LIN {X 0,Y 309.605,Z 177.893,A -85,B 0,C 180,E1 -15904.089,E2 -15904.089} C_VEL
LIN {X 0,Y 309.216,Z 180.991,A -85,B 0,C 180,E1 -15904.862,E2 -15904.862} C_VEL
LIN {X 0,Y 313.855,Z 215.016,A -85,B 0,C 180,E1 -15906.096,E2 -15906.096} C_VEL
LIN {X 0,Y 315.231,Z 227.724,A -85,B 0,C 180,E1 -15906.518,E2 -15906.518} C_VEL
LIN {X 0,Y 313.627,Z 290.842,A -85,B 0,C 180,E1 -15908.084,E2 -15908.084} C_VEL
LIN {X 0,Y 312.784,Z 304.258,A -85,B 0,C 180,E1 -15908.671,E2 -15908.671} C_VEL
LIN {X 0,Y 311.715,Z 316.542,A -85,B 0,C 180,E1 -15909.459,E2 -15909.459} C_VEL
LIN {X 0,Y 310.435,Z 328.402,A -85,B 0,C 180,E1 -15910.493,E2 -15910.493} C_VEL
LIN {X 0,Y 308.971,Z 339.839,A -85,B 0,C 180,E1 -15911.774,E2 -15911.774} C_VEL
LIN {X 0,Y 307.713,Z 350.2,A -85,B 0,C 180,E1 -15913.242,E2 -15913.242} C_VEL
LIN {X 0,Y 306.659,Z 358.857,A -85,B 0,C 180,E1 -15914.757,E2 -15914.757} C_VEL
LIN {X 0,Y 305.56,Z 367.859,A -85,B 0,C 180,E1 -15916.703,E2 -15916.703} C_VEL
LIN {X 0,Y 304.589,Z 375.237,A -85,B 0,C 180,E1 -15918.689,E2 -15918.689} C_VEL
LIN {X 0,Y 304.099,Z 381.144,A -85,B 0,C 180,E1 -15920.69,E2 -15920.69} C_VEL
LIN {X 0,Y 303.823,Z 385.764,A -85,B 0,C 180,E1 -15922.691,E2 -15922.691} C_VEL
LIN {X 0,Y 303.71,Z 389.249,A -85,B 0,C 180,E1 -15924.689,E2 -15924.689} C_VEL
LIN {X 0,Y 303.749,Z 390.973,A -85,B 0,C 180,E1 -15926.02,E2 -15926.02} C_VEL
LIN {X 0,Y 303.741,Z 392.268,A -85,B 0,C 180,E1 -15927.348,E2 -15927.348} C_VEL
LIN {X 0,Y 303.826,Z 393.159,A -85,B 0,C 180,E1 -15928.674,E2 -15928.674} C_VEL
LIN {X 0,Y 303.901,Z 393.618,A -85,B 0,C 180,E1 -15930,E2 -15930} C_VEL
LIN {X 0,Y 303.777,Z 393.629,A -85,B 0,C 180,E1 -15931.326,E2 -15931.326} C_VEL
LIN {X 0,Y 303.708,Z 393.245,A -85,B 0,C 180,E1 -15932.653,E2 -15932.653} C_VEL
LIN {X 0,Y 303.702,Z 392.469,A -85,B 0,C 180,E1 -15933.981,E2 -15933.981} C_VEL
LIN {X 0,Y 303.644,Z 390.958,A -85,B 0,C 180,E1 -15935.578,E2 -15935.578} C_VEL
LIN {X 0,Y 303.882,Z 387.555,A -85,B 0,C 180,E1 -15937.976,E2 -15937.976} C_VEL
LIN {X 0,Y 304.299,Z 383.584,A -85,B 0,C 180,E1 -15939.975,E2 -15939.975} C_VEL
LIN {X 0,Y 304.977,Z 378.484,A -85,B 0,C 180,E1 -15941.97,E2 -15941.97} C_VEL
LIN {X 0,Y 306.165,Z 372.114,A -85,B 0,C 180,E1 -15943.947,E2 -15943.947} C_VEL
LIN {X 0,Y 307.574,Z 364.197,A -85,B 0,C 180,E1 -15945.914,E2 -15945.914} C_VEL
LIN {X 0,Y 309.228,Z 354.358,A -85,B 0,C 180,E1 -15947.868,E2 -15947.868} C_VEL
LIN {X 0,Y 311.011,Z 344.245,A -85,B 0,C 180,E1 -15949.47,E2 -15949.47} C_VEL
LIN {X 0,Y 312.942,Z 332.854,A -85,B 0,C 180,E1 -15950.886,E2 -15950.886} C_VEL
LIN {X 0,Y 314.607,Z 321.762,A -85,B 0,C 180,E1 -15951.973,E2 -15951.973} C_VEL
LIN {X 0,Y 316.144,Z 309.533,A -85,B 0,C 180,E1 -15952.894,E2 -15952.894} C_VEL
LIN {X 0,Y 317.465,Z 296.002,A -85,B 0,C 180,E1 -15953.608,E2 -15953.608} C_VEL
LIN {X 0,Y 318.238,Z 283.152,A -85,B 0,C 180,E1 -15954.047,E2 -15954.047} C_VEL
LIN {X 0,Y 319.862,Z 226.172,A -85,B 0,C 180,E1 -15955.466,E2 -15955.466} C_VEL
LIN {X 0,Y 317.021,Z 205.398,A -85,B 0,C 180,E1 -15956.349,E2 -15956.349} C_VEL
LIN {X 0,Y 313.131,Z 184.639,A -85,B 0,C 180,E1 -15957.383,E2 -15957.383} C_VEL
LIN {X 0,Y 311.782,Z 178.357,A -85,B 0,C 180,E1 -15957.736,E2 -15957.736} C_VEL
LIN {X 0,Y 310.59,Z 171.052,A -85,B 0,C 180,E1 -15959.855,E2 -15959.855} C_VEL
LIN {X 0,Y 308.122,Z 160.384,A -85,B 0,C 180,E1 -15963.19,E2 -15963.19} C_VEL
LIN {X 0,Y 305.482,Z 150.438,A -85,B 0,C 180,E1 -15966.587,E2 -15966.587} C_VEL
LIN {X 0,Y 305.466,Z 150.444,A -85,B 0,C 180,E1 -15970.106,E2 -15970.106} C_VEL
LIN {X 0,Y 305.447,Z 150.439,A -85,B 0,C 180,E1 -15973.651,E2 -15973.651} C_VEL
LIN {X 0,Y 305.488,Z 150.436,A -85,B 0,C 180,E1 -15977.407,E2 -15977.407} C_VEL
LIN {X 0,Y 305.518,Z 150.425,A -85,B 0,C 180,E1 -15981.603,E2 -15981.603} C_VEL
LIN {X 0,Y 305.462,Z 150.434,A -85,B 0,C 180,E1 -15984.886,E2 -15984.886} C_VEL
LIN {X 0,Y 305.452,Z 150.437,A -85,B 0,C 180,E1 -15988.354,E2 -15988.354} C_VEL
LIN {X 0,Y 305.52,Z 150.422,A -85,B 0,C 180,E1 -15991.113,E2 -15991.113} C_VEL
LIN {X 0,Y 305.57,Z 150.414,A -85,B 0,C 180,E1 -15994.087,E2 -15994.087} C_VEL
LIN {X 0,Y 305.481,Z 150.428,A -85,B 0,C 180,E1 -15998.401,E2 -15998.401} C_VEL
LIN {X 0,Y 305.589,Z 150.41,A -85,B 0,C 180,E1 -16001.217,E2 -16001.217} C_VEL
LIN {X 0,Y 305.648,Z 150.404,A -85,B 0,C 180,E1 -16005.349,E2 -16005.349} C_VEL
LIN {X 0,Y 305.637,Z 150.408,A -85,B 0,C 180,E1 -16009.399,E2 -16009.399} C_VEL
LIN {X 0,Y 305.812,Z 150.385,A -85,B 0,C 180,E1 -16012.074,E2 -16012.074} C_VEL
LIN {X 0,Y 305.688,Z 150.408,A -85,B 0,C 180,E1 -16014.723,E2 -16014.723} C_VEL
LIN {X 0,Y 305.956,Z 150.373,A -85,B 0,C 180,E1 -16018.683,E2 -16018.683} C_VEL
LIN {X 0,Y 305.956,Z 150.375,A -85,B 0,C 180,E1 -16021.316,E2 -16021.316} C_VEL
LIN {X 0,Y 305.685,Z 150.405,A -85,B 0,C 180,E1 -16025.276,E2 -16025.276} C_VEL
LIN {X 0,Y 305.795,Z 150.394,A -85,B 0,C 180,E1 -16027.926,E2 -16027.926} C_VEL
LIN {X 0,Y 305.602,Z 150.416,A -85,B 0,C 180,E1 -16031.945,E2 -16031.945} C_VEL
LIN {X 0,Y 305.636,Z 150.417,A -85,B 0,C 180,E1 -16035.035,E2 -16035.035} C_VEL
LIN {X 0,Y 305.575,Z 150.422,A -85,B 0,C 180,E1 -16039.445,E2 -16039.445} C_VEL
LIN {X 0,Y 305.527,Z 150.521,A -85,B 0,C 180,E1 -16044.062,E2 -16044.062} C_VEL
LIN {X 0,Y 306.019,Z 152.265,A -85,B 0,C 180,E1 -16044.643,E2 -16044.643} C_VEL
LIN {X 0,Y 313.705,Z 166.916,A -85,B 0,C 180,E1 -16046.023,E2 -16046.023} C_VEL
LIN {X 0,Y 320.196,Z 181.578,A -85,B 0,C 180,E1 -16047.174,E2 -16047.174} C_VEL
LIN {X 0,Y 321.198,Z 184.098,A -85,B 0,C 180,E1 -16047.354,E2 -16047.354} C_VEL
LIN {X 0,Y 318.681,Z 259.47,A -85,B 0,C 180,E1 -16049.25,E2 -16049.25} C_VEL
LIN {X 0,Y 317.9,Z 272.399,A -85,B 0,C 180,E1 -16049.829,E2 -16049.829} C_VEL
LIN {X 0,Y 316.94,Z 283.918,A -85,B 0,C 180,E1 -16050.574,E2 -16050.574} C_VEL
LIN {X 0,Y 315.772,Z 295.122,A -85,B 0,C 180,E1 -16051.535,E2 -16051.535} C_VEL
LIN {X 0,Y 314.394,Z 305.267,A -85,B 0,C 180,E1 -16052.635,E2 -16052.635} C_VEL
LIN {X 0,Y 312.641,Z 316.622,A -85,B 0,C 180,E1 -16054.193,E2 -16054.193} C_VEL
LIN {X 0,Y 310.868,Z 326.385,A -85,B 0,C 180,E1 -16055.868,E2 -16055.868} C_VEL
LIN {X 0,Y 309.235,Z 334.779,A -85,B 0,C 180,E1 -16057.68,E2 -16057.68} C_VEL
LIN {X 0,Y 307.645,Z 342.494,A -85,B 0,C 180,E1 -16059.765,E2 -16059.765} C_VEL
LIN {X 0,Y 306.527,Z 348.078,A -85,B 0,C 180,E1 -16061.675,E2 -16061.675} C_VEL
LIN {X 0,Y 305.613,Z 352.558,A -85,B 0,C 180,E1 -16063.621,E2 -16063.621} C_VEL
LIN {X 0,Y 304.652,Z 356.866,A -85,B 0,C 180,E1 -16066.206,E2 -16066.206} C_VEL
LIN {X 0,Y 304.229,Z 358.833,A -85,B 0,C 180,E1 -16067.939,E2 -16067.939} C_VEL
LIN {X 0,Y 303.894,Z 360.092,A -85,B 0,C 180,E1 -16069.744,E2 -16069.744} C_VEL
LIN {X 0,Y 303.659,Z 360.636,A -85,B 0,C 180,E1 -16071.897,E2 -16071.897} C_VEL
LIN {X 0,Y 303.648,Z 360.102,A -85,B 0,C 180,E1 -16074.104,E2 -16074.104} C_VEL
LIN {X 0,Y 303.839,Z 358.382,A -85,B 0,C 180,E1 -16076.377,E2 -16076.377} C_VEL
LIN {X 0,Y 304.229,Z 355.273,A -85,B 0,C 180,E1 -16078.73,E2 -16078.73} C_VEL
LIN {X 0,Y 304.763,Z 350.855,A -85,B 0,C 180,E1 -16081.036,E2 -16081.036} C_VEL
LIN {X 0,Y 305.446,Z 345.271,A -85,B 0,C 180,E1 -16083.215,E2 -16083.215} C_VEL
LIN {X 0,Y 306.369,Z 338.545,A -85,B 0,C 180,E1 -16085.251,E2 -16085.251} C_VEL
LIN {X 0,Y 307.411,Z 330.797,A -85,B 0,C 180,E1 -16087.13,E2 -16087.13} C_VEL
LIN {X 0,Y 308.685,Z 321.324,A -85,B 0,C 180,E1 -16088.982,E2 -16088.982} C_VEL
LIN {X 0,Y 309.814,Z 312.005,A -85,B 0,C 180,E1 -16090.452,E2 -16090.452} C_VEL
LIN {X 0,Y 311.123,Z 300.466,A -85,B 0,C 180,E1 -16091.905,E2 -16091.905} C_VEL
LIN {X 0,Y 312.261,Z 288.683,A -85,B 0,C 180,E1 -16093.071,E2 -16093.071} C_VEL
LIN {X 0,Y 313.041,Z 277.074,A -85,B 0,C 180,E1 -16093.953,E2 -16093.953} C_VEL
LIN {X 0,Y 313.833,Z 263.312,A -85,B 0,C 180,E1 -16094.692,E2 -16094.692} C_VEL
LIN {X 0,Y 314.307,Z 250.807,A -85,B 0,C 180,E1 -16095.114,E2 -16095.114} C_VEL
LIN {X 0,Y 316.167,Z 179.057,A -85,B 0,C 180,E1 -16096.847,E2 -16096.847} C_VEL
LIN {X 0,Y 308.843,Z 158.463,A -85,B 0,C 180,E1 -16097.91,E2 -16097.91} C_VEL
LIN {X 0,Y 305.699,Z 150.706,A -85,B 0,C 180,E1 -16098.353,E2 -16098.353} C_VEL
LIN {X 0,Y 305.635,Z 150.414,A -85,B 0,C 180,E1 -16098.393,E2 -16098.393} C_VEL
LIN {X 0,Y 305.8,Z 150.394,A -85,B 0,C 180,E1 -16102.074,E2 -16102.074} C_VEL
LIN {X 0,Y 305.685,Z 150.406,A -85,B 0,C 180,E1 -16104.723,E2 -16104.723} C_VEL
LIN {X 0,Y 305.955,Z 150.372,A -85,B 0,C 180,E1 -16108.684,E2 -16108.684} C_VEL
LIN {X 0,Y 305.955,Z 150.377,A -85,B 0,C 180,E1 -16111.316,E2 -16111.316} C_VEL
LIN {X 0,Y 305.674,Z 150.411,A -85,B 0,C 180,E1 -16115.277,E2 -16115.277} C_VEL
LIN {X 0,Y 305.749,Z 150.398,A -85,B 0,C 180,E1 -16117.927,E2 -16117.927} C_VEL
LIN {X 0,Y 305.599,Z 150.416,A -85,B 0,C 180,E1 -16121.945,E2 -16121.945} C_VEL
LIN {X 0,Y 305.608,Z 150.419,A -85,B 0,C 180,E1 -16125.015,E2 -16125.015} C_VEL
LIN {X 0,Y 305.541,Z 150.424,A -85,B 0,C 180,E1 -16129.426,E2 -16129.426} C_VEL
LIN {X 0,Y 305.485,Z 150.432,A -85,B 0,C 180,E1 -16133.039,E2 -16133.039} C_VEL
LIN {X 0,Y 305.553,Z 150.423,A -85,B 0,C 180,E1 -16136.229,E2 -16136.229} C_VEL
LIN {X 0,Y 305.495,Z 150.43,A -85,B 0,C 180,E1 -16139.05,E2 -16139.05} C_VEL
LIN {X 0,Y 305.464,Z 150.432,A -85,B 0,C 180,E1 -16143.517,E2 -16143.517} C_VEL
LIN {X 0,Y 305.473,Z 150.434,A -85,B 0,C 180,E1 -16146.739,E2 -16146.739} C_VEL
LIN {X 0,Y 305.453,Z 150.434,A -85,B 0,C 180,E1 -16150.6,E2 -16150.6} C_VEL
LIN {X 0,Y 305.424,Z 150.437,A -85,B 0,C 180,E1 -16153.655,E2 -16153.655} C_VEL
LIN {X 0,Y 305.453,Z 150.433,A -85,B 0,C 180,E1 -16157.414,E2 -16157.414} C_VEL
LIN {X 0,Y 305.448,Z 150.431,A -85,B 0,C 180,E1 -16161.215,E2 -16161.215} C_VEL
LIN {X 0,Y 304.815,Z 150.516,A -85,B 0,C 180,E1 -16162.315,E2 -16162.315} C_VEL
LIN {X 0,Y 301.928,Z 150.877,A -85,B 0,C 180,E1 -16164.104,E2 -16164.104} C_VEL
LIN {X 0,Y 299.474,Z 151.18,A -85,B 0,C 180,E1 -16165.556,E2 -16165.556} C_VEL
LIN {X 0,Y 298.451,Z 151.306,A -85,B 0,C 180,E1 -16166.682,E2 -16166.682} C_VEL
LIN {X 0,Y 298.386,Z 151.313,A -85,B 0,C 180,E1 -16167.063,E2 -16167.063} C_VEL
LIN {X 0,Y 298.43,Z 151.304,A -85,B 0,C 180,E1 -16170.615,E2 -16170.615} C_VEL
LIN {X 0,Y 298.482,Z 151.303,A -85,B 0,C 180,E1 -16173.474,E2 -16173.474} C_VEL
LIN {X 0,Y 298.429,Z 151.309,A -85,B 0,C 180,E1 -16176.7,E2 -16176.7} C_VEL
LIN {X 0,Y 298.537,Z 151.293,A -85,B 0,C 180,E1 -16180.757,E2 -16180.757} C_VEL
LIN {X 0,Y 298.592,Z 151.288,A -85,B 0,C 180,E1 -16184.995,E2 -16184.995} C_VEL
LIN {X 0,Y 298.593,Z 151.291,A -85,B 0,C 180,E1 -16189.147,E2 -16189.147} C_VEL
LIN {X 0,Y 298.757,Z 151.266,A -85,B 0,C 180,E1 -16191.886,E2 -16191.886} C_VEL
LIN {X 0,Y 298.659,Z 151.277,A -85,B 0,C 180,E1 -16194.599,E2 -16194.599} C_VEL
LIN {X 0,Y 298.923,Z 151.248,A -85,B 0,C 180,E1 -16198.653,E2 -16198.653} C_VEL
LIN {X 0,Y 298.923,Z 151.248,A -85,B 0,C 180,E1 -16201.348,E2 -16201.348} C_VEL
LIN {X 0,Y 298.791,Z 151.266,A -85,B 0,C 180,E1 -16206.754,E2 -16206.754} C_VEL
LIN {X 0,Y 298.68,Z 151.277,A -85,B 0,C 180,E1 -16209.481,E2 -16209.481} C_VEL
LIN {X 0,Y 298.551,Z 151.292,A -85,B 0,C 180,E1 -16213.616,E2 -16213.616} C_VEL
LIN {X 0,Y 298.548,Z 151.296,A -85,B 0,C 180,E1 -16216.409,E2 -16216.409} C_VEL
LIN {X 0,Y 298.51,Z 151.297,A -85,B 0,C 180,E1 -16219.654,E2 -16219.654} C_VEL
LIN {X 0,Y 298.428,Z 151.309,A -85,B 0,C 180,E1 -16223.6,E2 -16223.6} C_VEL
LIN {X 0,Y 298.489,Z 151.304,A -85,B 0,C 180,E1 -16226.575,E2 -16226.575} C_VEL
LIN {X 0,Y 298.421,Z 151.311,A -85,B 0,C 180,E1 -16229.641,E2 -16229.641} C_VEL
LIN {X 0,Y 298.396,Z 151.314,A -85,B 0,C 180,E1 -16232.801,E2 -16232.801} C_VEL
LIN {X 0,Y 298.466,Z 151.305,A -85,B 0,C 180,E1 -16236.813,E2 -16236.813} C_VEL
LIN {X 0,Y 298.418,Z 151.311,A -85,B 0,C 180,E1 -16241.095,E2 -16241.095} C_VEL
LIN {X 0,Y 298.427,Z 151.309,A -85,B 0,C 180,E1 -16243.109,E2 -16243.109} C_VEL
LIN {X 0,Y 298.433,Z 151.308,A -85,B 0,C 180,E1 -16246.926,E2 -16246.926} C_VEL
LIN {X 0,Y 298.432,Z 151.31,A -85,B 0,C 180,E1 -16251,E2 -16251} C_VEL
LIN {X 0,Y 298.434,Z 151.312,A -85,B 0,C 180,E1 -16253.933,E2 -16253.933} C_VEL
LIN {X 0,Y 298.472,Z 151.434,A -85,B 0,C 180,E1 -16256.099,E2 -16256.099} C_VEL
LIN {X 0,Y 301.505,Z 165.405,A -85,B 0,C 180,E1 -16260.229,E2 -16260.229} C_VEL
LIN {X 0,Y 303.03,Z 172.939,A -85,B 0,C 180,E1 -16262.364,E2 -16262.364} C_VEL
LIN {X 0,Y 302.835,Z 177.137,A -85,B 0,C 180,E1 -16263.465,E2 -16263.465} C_VEL
LIN {X 0,Y 302.407,Z 180.637,A -85,B 0,C 180,E1 -16264.362,E2 -16264.362} C_VEL
LIN {X 0,Y 307.043,Z 214.787,A -85,B 0,C 180,E1 -16265.636,E2 -16265.636} C_VEL
LIN {X 0,Y 308.549,Z 227.299,A -85,B 0,C 180,E1 -16266.074,E2 -16266.074} C_VEL
LIN {X 0,Y 306.907,Z 290.169,A -85,B 0,C 180,E1 -16267.667,E2 -16267.667} C_VEL
LIN {X 0,Y 306.041,Z 303.671,A -85,B 0,C 180,E1 -16268.266,E2 -16268.266} C_VEL
LIN {X 0,Y 304.907,Z 316.005,A -85,B 0,C 180,E1 -16269.067,E2 -16269.067} C_VEL
LIN {X 0,Y 303.528,Z 328.703,A -85,B 0,C 180,E1 -16270.206,E2 -16270.206} C_VEL
LIN {X 0,Y 302.023,Z 340.017,A -85,B 0,C 180,E1 -16271.515,E2 -16271.515} C_VEL
LIN {X 0,Y 300.732,Z 350.248,A -85,B 0,C 180,E1 -16273.015,E2 -16273.015} C_VEL
LIN {X 0,Y 299.553,Z 359.788,A -85,B 0,C 180,E1 -16274.761,E2 -16274.761} C_VEL
LIN {X 0,Y 298.406,Z 368.461,A -85,B 0,C 180,E1 -16276.725,E2 -16276.725} C_VEL
LIN {X 0,Y 297.459,Z 375.637,A -85,B 0,C 180,E1 -16278.76,E2 -16278.76} C_VEL
LIN {X 0,Y 296.946,Z 382.182,A -85,B 0,C 180,E1 -16281.151,E2 -16281.151} C_VEL
LIN {X 0,Y 296.702,Z 386.466,A -85,B 0,C 180,E1 -16283.198,E2 -16283.198} C_VEL
LIN {X 0,Y 296.642,Z 388.725,A -85,B 0,C 180,E1 -16284.562,E2 -16284.562} C_VEL
LIN {X 0,Y 296.657,Z 390.484,A -85,B 0,C 180,E1 -16285.924,E2 -16285.924} C_VEL
LIN {X 0,Y 296.661,Z 391.803,A -85,B 0,C 180,E1 -16287.284,E2 -16287.284} C_VEL
LIN {X 0,Y 296.732,Z 392.714,A -85,B 0,C 180,E1 -16288.643,E2 -16288.643} C_VEL
LIN {X 0,Y 296.811,Z 393.211,A -85,B 0,C 180,E1 -16290,E2 -16290} C_VEL
LIN {X 0,Y 296.685,Z 393.246,A -85,B 0,C 180,E1 -16291.357,E2 -16291.357} C_VEL
LIN {X 0,Y 296.628,Z 392.883,A -85,B 0,C 180,E1 -16292.716,E2 -16292.716} C_VEL
LIN {X 0,Y 296.61,Z 392.125,A -85,B 0,C 180,E1 -16294.076,E2 -16294.076} C_VEL
LIN {X 0,Y 296.547,Z 390.884,A -85,B 0,C 180,E1 -16295.508,E2 -16295.508} C_VEL
LIN {X 0,Y 296.827,Z 387.29,A -85,B 0,C 180,E1 -16298.167,E2 -16298.167} C_VEL
LIN {X 0,Y 297.269,Z 383.361,A -85,B 0,C 180,E1 -16300.213,E2 -16300.213} C_VEL
LIN {X 0,Y 297.999,Z 378.311,A -85,B 0,C 180,E1 -16302.254,E2 -16302.254} C_VEL
LIN {X 0,Y 299.262,Z 372.009,A -85,B 0,C 180,E1 -16304.275,E2 -16304.275} C_VEL
LIN {X 0,Y 300.745,Z 364.208,A -85,B 0,C 180,E1 -16306.285,E2 -16306.285} C_VEL
LIN {X 0,Y 302.141,Z 356.263,A -85,B 0,C 180,E1 -16307.951,E2 -16307.951} C_VEL
LIN {X 0,Y 304.123,Z 345.536,A -85,B 0,C 180,E1 -16309.753,E2 -16309.753} C_VEL
LIN {X 0,Y 306.153,Z 334.655,A -85,B 0,C 180,E1 -16311.195,E2 -16311.195} C_VEL
LIN {X 0,Y 308.052,Z 322.344,A -85,B 0,C 180,E1 -16312.466,E2 -16312.466} C_VEL
LIN {X 0,Y 309.805,Z 309.277,A -85,B 0,C 180,E1 -16313.479,E2 -16313.479} C_VEL
LIN {X 0,Y 311.174,Z 295.74,A -85,B 0,C 180,E1 -16314.209,E2 -16314.209} C_VEL
LIN {X 0,Y 311.981,Z 282.408,A -85,B 0,C 180,E1 -16314.674,E2 -16314.674} C_VEL
LIN {X 0,Y 313.717,Z 227.416,A -85,B 0,C 180,E1 -16316.069,E2 -16316.069} C_VEL
LIN {X 0,Y 310.987,Z 206.911,A -85,B 0,C 180,E1 -16316.971,E2 -16316.971} C_VEL
LIN {X 0,Y 307.427,Z 187.646,A -85,B 0,C 180,E1 -16317.958,E2 -16317.958} C_VEL
LIN {X 0,Y 305.766,Z 180.708,A -85,B 0,C 180,E1 -16318.374,E2 -16318.374} C_VEL
LIN {X 0,Y 304.746,Z 177.782,A -85,B 0,C 180,E1 -16318.619,E2 -16318.619} C_VEL
LIN {X 0,Y 302.538,Z 167.202,A -85,B 0,C 180,E1 -16321.903,E2 -16321.903} C_VEL
LIN {X 0,Y 300.04,Z 157.167,A -85,B 0,C 180,E1 -16325.272,E2 -16325.272} C_VEL
LIN {X 0,Y 298.434,Z 151.316,A -85,B 0,C 180,E1 -16327.423,E2 -16327.423} C_VEL
LIN {X 0,Y 298.419,Z 151.316,A -85,B 0,C 180,E1 -16331.255,E2 -16331.255} C_VEL
LIN {X 0,Y 298.36,Z 151.324,A -85,B 0,C 180,E1 -16334.964,E2 -16334.964} C_VEL
LIN {X 0,Y 298.432,Z 151.315,A -85,B 0,C 180,E1 -16336.926,E2 -16336.926} C_VEL
LIN {X 0,Y 298.431,Z 151.307,A -85,B 0,C 180,E1 -16340.999,E2 -16340.999} C_VEL
LIN {X 0,Y 298.433,Z 151.306,A -85,B 0,C 180,E1 -16343.932,E2 -16343.932} C_VEL
LIN {X 0,Y 298.395,Z 151.313,A -85,B 0,C 180,E1 -16347.983,E2 -16347.983} C_VEL
LIN {X 0,Y 298.463,Z 151.308,A -85,B 0,C 180,E1 -16351.904,E2 -16351.904} C_VEL
LIN {X 0,Y 298.483,Z 151.299,A -85,B 0,C 180,E1 -16354.923,E2 -16354.923} C_VEL
LIN {X 0,Y 298.439,Z 151.308,A -85,B 0,C 180,E1 -16359.314,E2 -16359.314} C_VEL
LIN {X 0,Y 298.537,Z 151.294,A -85,B 0,C 180,E1 -16362.179,E2 -16362.179} C_VEL
LIN {X 0,Y 298.592,Z 151.282,A -85,B 0,C 180,E1 -16364.994,E2 -16364.994} C_VEL
LIN {X 0,Y 298.592,Z 151.283,A -85,B 0,C 180,E1 -16369.146,E2 -16369.146} C_VEL
LIN {X 0,Y 298.757,Z 151.265,A -85,B 0,C 180,E1 -16371.886,E2 -16371.886} C_VEL
LIN {X 0,Y 298.659,Z 151.283,A -85,B 0,C 180,E1 -16374.599,E2 -16374.599} C_VEL
LIN {X 0,Y 298.922,Z 151.249,A -85,B 0,C 180,E1 -16378.652,E2 -16378.652} C_VEL
LIN {X 0,Y 298.922,Z 151.251,A -85,B 0,C 180,E1 -16381.347,E2 -16381.347} C_VEL
LIN {X 0,Y 298.785,Z 151.264,A -85,B 0,C 180,E1 -16386.754,E2 -16386.754} C_VEL
LIN {X 0,Y 298.634,Z 151.285,A -85,B 0,C 180,E1 -16389.482,E2 -16389.482} C_VEL
LIN {X 0,Y 298.55,Z 151.295,A -85,B 0,C 180,E1 -16393.615,E2 -16393.615} C_VEL
LIN {X 0,Y 298.547,Z 151.295,A -85,B 0,C 180,E1 -16396.408,E2 -16396.408} C_VEL
LIN {X 0,Y 298.51,Z 151.301,A -85,B 0,C 180,E1 -16399.655,E2 -16399.655} C_VEL
LIN {X 0,Y 298.494,Z 151.402,A -85,B 0,C 180,E1 -16403.26,E2 -16403.26} C_VEL
LIN {X 0,Y 298.694,Z 152.48,A -85,B 0,C 180,E1 -16403.669,E2 -16403.669} C_VEL
LIN {X 0,Y 306.611,Z 167.127,A -85,B 0,C 180,E1 -16405.181,E2 -16405.181} C_VEL
LIN {X 0,Y 312.778,Z 180.395,A -85,B 0,C 180,E1 -16406.314,E2 -16406.314} C_VEL
LIN {X 0,Y 315.128,Z 186.194,A -85,B 0,C 180,E1 -16406.75,E2 -16406.75} C_VEL
LIN {X 0,Y 312.456,Z 259.797,A -85,B 0,C 180,E1 -16408.638,E2 -16408.638} C_VEL
LIN {X 0,Y 311.609,Z 272.96,A -85,B 0,C 180,E1 -16409.24,E2 -16409.24} C_VEL
LIN {X 0,Y 310.501,Z 285.544,A -85,B 0,C 180,E1 -16410.086,E2 -16410.086} C_VEL
LIN {X 0,Y 309.168,Z 297.063,A -85,B 0,C 180,E1 -16411.129,E2 -16411.129} C_VEL
LIN {X 0,Y 307.494,Z 308.603,A -85,B 0,C 180,E1 -16412.465,E2 -16412.465} C_VEL
LIN {X 0,Y 305.806,Z 318.7,A -85,B 0,C 180,E1 -16413.939,E2 -16413.939} C_VEL
LIN {X 0,Y 304.054,Z 327.766,A -85,B 0,C 180,E1 -16415.585,E2 -16415.585} C_VEL
LIN {X 0,Y 302.35,Z 336.001,A -85,B 0,C 180,E1 -16417.435,E2 -16417.435} C_VEL
LIN {X 0,Y 300.736,Z 343.483,A -85,B 0,C 180,E1 -16419.54,E2 -16419.54} C_VEL
LIN {X 0,Y 299.378,Z 349.659,A -85,B 0,C 180,E1 -16421.795,E2 -16421.795} C_VEL
LIN {X 0,Y 298.329,Z 354.37,A -85,B 0,C 180,E1 -16424.068,E2 -16424.068} C_VEL
LIN {X 0,Y 297.418,Z 358.234,A -85,B 0,C 180,E1 -16426.744,E2 -16426.744} C_VEL
LIN {X 0,Y 296.875,Z 360.309,A -85,B 0,C 180,E1 -16429.248,E2 -16429.248} C_VEL
LIN {X 0,Y 296.581,Z 361.042,A -85,B 0,C 180,E1 -16431.967,E2 -16431.967} C_VEL
LIN {X 0,Y 296.553,Z 360.638,A -85,B 0,C 180,E1 -16433.684,E2 -16433.684} C_VEL
LIN {X 0,Y 296.692,Z 359.105,A -85,B 0,C 180,E1 -16436.003,E2 -16436.003} C_VEL
LIN {X 0,Y 297.114,Z 355.879,A -85,B 0,C 180,E1 -16438.642,E2 -16438.642} C_VEL
LIN {X 0,Y 297.647,Z 351.78,A -85,B 0,C 180,E1 -16440.884,E2 -16440.884} C_VEL
LIN {X 0,Y 298.423,Z 345.503,A -85,B 0,C 180,E1 -16443.419,E2 -16443.419} C_VEL
LIN {X 0,Y 299.46,Z 338.296,A -85,B 0,C 180,E1 -16445.617,E2 -16445.617} C_VEL
LIN {X 0,Y 300.658,Z 329.79,A -85,B 0,C 180,E1 -16447.676,E2 -16447.676} C_VEL
LIN {X 0,Y 301.797,Z 321.404,A -85,B 0,C 180,E1 -16449.316,E2 -16449.316} C_VEL
LIN {X 0,Y 303.032,Z 311.571,A -85,B 0,C 180,E1 -16450.878,E2 -16450.878} C_VEL
LIN {X 0,Y 304.394,Z 299.598,A -85,B 0,C 180,E1 -16452.392,E2 -16452.392} C_VEL
LIN {X 0,Y 305.566,Z 287.769,A -85,B 0,C 180,E1 -16453.55,E2 -16453.55} C_VEL
LIN {X 0,Y 306.407,Z 275.87,A -85,B 0,C 180,E1 -16454.438,E2 -16454.438} C_VEL
LIN {X 0,Y 307.155,Z 262.7,A -85,B 0,C 180,E1 -16455.138,E2 -16455.138} C_VEL
LIN {X 0,Y 307.641,Z 249.064,A -85,B 0,C 180,E1 -16455.577,E2 -16455.577} C_VEL
LIN {X 0,Y 309.367,Z 180.053,A -85,B 0,C 180,E1 -16457.291,E2 -16457.291} C_VEL
LIN {X 0,Y 302.107,Z 159.981,A -85,B 0,C 180,E1 -16458.369,E2 -16458.369} C_VEL
LIN {X 0,Y 298.761,Z 152.111,A -85,B 0,C 180,E1 -16458.844,E2 -16458.844} C_VEL
LIN {X 0,Y 298.612,Z 151.29,A -85,B 0,C 180,E1 -16458.916,E2 -16458.916} C_VEL
LIN {X 0,Y 298.745,Z 151.274,A -85,B 0,C 180,E1 -16461.886,E2 -16461.886} C_VEL
LIN {X 0,Y 298.656,Z 151.282,A -85,B 0,C 180,E1 -16464.599,E2 -16464.599} C_VEL
LIN {X 0,Y 298.922,Z 151.248,A -85,B 0,C 180,E1 -16468.653,E2 -16468.653} C_VEL
LIN {X 0,Y 298.922,Z 151.253,A -85,B 0,C 180,E1 -16471.347,E2 -16471.347} C_VEL
LIN {X 0,Y 298.642,Z 151.287,A -85,B 0,C 180,E1 -16475.401,E2 -16475.401} C_VEL
LIN {X 0,Y 298.708,Z 151.277,A -85,B 0,C 180,E1 -16478.821,E2 -16478.821} C_VEL
LIN {X 0,Y 298.545,Z 151.295,A -85,B 0,C 180,E1 -16483.616,E2 -16483.616} C_VEL
LIN {X 0,Y 298.486,Z 151.303,A -85,B 0,C 180,E1 -16486.412,E2 -16486.412} C_VEL
LIN {X 0,Y 298.482,Z 151.302,A -85,B 0,C 180,E1 -16489.639,E2 -16489.639} C_VEL
LIN {X 0,Y 298.428,Z 151.308,A -85,B 0,C 180,E1 -16493.6,E2 -16493.6} C_VEL
LIN {X 0,Y 298.491,Z 151.305,A -85,B 0,C 180,E1 -16496.574,E2 -16496.574} C_VEL
LIN {X 0,Y 298.42,Z 151.31,A -85,B 0,C 180,E1 -16499.641,E2 -16499.641} C_VEL
LIN {X 0,Y 298.394,Z 151.316,A -85,B 0,C 180,E1 -16502.8,E2 -16502.8} C_VEL
LIN {X 0,Y 298.445,Z 151.309,A -85,B 0,C 180,E1 -16506.808,E2 -16506.808} C_VEL
LIN {X 0,Y 298.385,Z 151.311,A -85,B 0,C 180,E1 -16511.088,E2 -16511.088} C_VEL
LIN {X 0,Y 298.397,Z 151.312,A -85,B 0,C 180,E1 -16513.103,E2 -16513.103} C_VEL
LIN {X 0,Y 298.401,Z 151.312,A -85,B 0,C 180,E1 -16516.921,E2 -16516.921} C_VEL
LIN {X 0,Y 298.406,Z 151.308,A -85,B 0,C 180,E1 -16521.207,E2 -16521.207} C_VEL
LIN {X 0,Y 298.419,Z 151.313,A -85,B 0,C 180,E1 -16523.931,E2 -16523.931} C_VEL
LIN {X 0,Y 298.386,Z 151.313,A -85,B 0,C 180,E1 -16527.063,E2 -16527.063} C_VEL
LIN {X 0,Y 297.763,Z 151.396,A -85,B 0,C 180,E1 -16528.19,E2 -16528.19} C_VEL
LIN {X 0,Y 294.92,Z 151.748,A -85,B 0,C 180,E1 -16530.026,E2 -16530.026} C_VEL
LIN {X 0,Y 292.503,Z 152.045,A -85,B 0,C 180,E1 -16531.516,E2 -16531.516} C_VEL
LIN {X 0,Y 291.497,Z 152.17,A -85,B 0,C 180,E1 -16532.67,E2 -16532.67} C_VEL
LIN {X 0,Y 291.434,Z 152.178,A -85,B 0,C 180,E1 -16533.061,E2 -16533.061} C_VEL
LIN {X 0,Y 291.373,Z 152.19,A -85,B 0,C 180,E1 -16537.299,E2 -16537.299} C_VEL
LIN {X 0,Y 291.457,Z 152.175,A -85,B 0,C 180,E1 -16540.27,E2 -16540.27} C_VEL
LIN {X 0,Y 291.554,Z 152.163,A -85,B 0,C 180,E1 -16544.624,E2 -16544.624} C_VEL
LIN {X 0,Y 291.536,Z 152.168,A -85,B 0,C 180,E1 -16548.881,E2 -16548.881} C_VEL
LIN {X 0,Y 291.708,Z 152.144,A -85,B 0,C 180,E1 -16551.689,E2 -16551.689} C_VEL
LIN {X 0,Y 291.63,Z 152.152,A -85,B 0,C 180,E1 -16554.469,E2 -16554.469} C_VEL
LIN {X 0,Y 291.889,Z 152.124,A -85,B 0,C 180,E1 -16558.621,E2 -16558.621} C_VEL
LIN {X 0,Y 291.889,Z 152.123,A -85,B 0,C 180,E1 -16561.38,E2 -16561.38} C_VEL
LIN {X 0,Y 291.74,Z 152.145,A -85,B 0,C 180,E1 -16566.918,E2 -16566.918} C_VEL
LIN {X 0,Y 291.629,Z 152.155,A -85,B 0,C 180,E1 -16569.712,E2 -16569.712} C_VEL
LIN {X 0,Y 291.521,Z 152.168,A -85,B 0,C 180,E1 -16573.951,E2 -16573.951} C_VEL
LIN {X 0,Y 291.487,Z 152.177,A -85,B 0,C 180,E1 -16576.818,E2 -16576.818} C_VEL
LIN {X 0,Y 291.45,Z 152.176,A -85,B 0,C 180,E1 -16579.875,E2 -16579.875} C_VEL
LIN {X 0,Y 291.383,Z 152.189,A -85,B 0,C 180,E1 -16584.207,E2 -16584.207} C_VEL
LIN {X 0,Y 291.423,Z 152.181,A -85,B 0,C 180,E1 -16587.272,E2 -16587.272} C_VEL
LIN {X 0,Y 291.337,Z 152.196,A -85,B 0,C 180,E1 -16590.437,E2 -16590.437} C_VEL
LIN {X 0,Y 291.345,Z 152.192,A -85,B 0,C 180,E1 -16593.699,E2 -16593.699} C_VEL
LIN {X 0,Y 291.401,Z 152.184,A -85,B 0,C 180,E1 -16597.261,E2 -16597.261} C_VEL
LIN {X 0,Y 291.377,Z 152.189,A -85,B 0,C 180,E1 -16600.635,E2 -16600.635} C_VEL
LIN {X 0,Y 291.302,Z 152.198,A -85,B 0,C 180,E1 -16604.4,E2 -16604.4} C_VEL
LIN {X 0,Y 291.356,Z 152.192,A -85,B 0,C 180,E1 -16608.398,E2 -16608.398} C_VEL
LIN {X 0,Y 291.382,Z 152.189,A -85,B 0,C 180,E1 -16611.163,E2 -16611.163} C_VEL
LIN {X 0,Y 291.387,Z 152.188,A -85,B 0,C 180,E1 -16614.63,E2 -16614.63} C_VEL
LIN {X 0,Y 291.409,Z 152.396,A -85,B 0,C 180,E1 -16615.705,E2 -16615.705} C_VEL
LIN {X 0,Y 294.05,Z 164.401,A -85,B 0,C 180,E1 -16619.365,E2 -16619.365} C_VEL
LIN {X 0,Y 295.946,Z 173.524,A -85,B 0,C 180,E1 -16622.03,E2 -16622.03} C_VEL
LIN {X 0,Y 296.103,Z 176.358,A -85,B 0,C 180,E1 -16622.813,E2 -16622.813} C_VEL
LIN {X 0,Y 295.599,Z 180.238,A -85,B 0,C 180,E1 -16623.83,E2 -16623.83} C_VEL
LIN {X 0,Y 300.386,Z 215.514,A -85,B 0,C 180,E1 -16625.192,E2 -16625.192} C_VEL
LIN {X 0,Y 301.821,Z 228.349,A -85,B 0,C 180,E1 -16625.646,E2 -16625.646} C_VEL
LIN {X 0,Y 300.191,Z 289.491,A -85,B 0,C 180,E1 -16627.231,E2 -16627.231} C_VEL
LIN {X 0,Y 299.302,Z 303.08,A -85,B 0,C 180,E1 -16627.842,E2 -16627.842} C_VEL
LIN {X 0,Y 298.145,Z 315.473,A -85,B 0,C 180,E1 -16628.66,E2 -16628.66} C_VEL
LIN {X 0,Y 296.806,Z 327.414,A -85,B 0,C 180,E1 -16629.739,E2 -16629.739} C_VEL
LIN {X 0,Y 295.306,Z 338.902,A -85,B 0,C 180,E1 -16631.079,E2 -16631.079} C_VEL
LIN {X 0,Y 293.918,Z 349.293,A -85,B 0,C 180,E1 -16632.609,E2 -16632.609} C_VEL
LIN {X 0,Y 292.593,Z 359.147,A -85,B 0,C 180,E1 -16634.436,E2 -16634.436} C_VEL
LIN {X 0,Y 291.462,Z 367.691,A -85,B 0,C 180,E1 -16636.402,E2 -16636.402} C_VEL
LIN {X 0,Y 290.451,Z 374.958,A -85,B 0,C 180,E1 -16638.485,E2 -16638.485} C_VEL
LIN {X 0,Y 290.018,Z 379.867,A -85,B 0,C 180,E1 -16640.234,E2 -16640.234} C_VEL
LIN {X 0,Y 289.698,Z 384.607,A -85,B 0,C 180,E1 -16642.332,E2 -16642.332} C_VEL
LIN {X 0,Y 289.56,Z 388.19,A -85,B 0,C 180,E1 -16644.429,E2 -16644.429} C_VEL
LIN {X 0,Y 289.57,Z 389.995,A -85,B 0,C 180,E1 -16645.824,E2 -16645.824} C_VEL
LIN {X 0,Y 289.583,Z 391.337,A -85,B 0,C 180,E1 -16647.218,E2 -16647.218} C_VEL
LIN {X 0,Y 289.64,Z 392.269,A -85,B 0,C 180,E1 -16648.61,E2 -16648.61} C_VEL
LIN {X 0,Y 289.721,Z 392.796,A -85,B 0,C 180,E1 -16650,E2 -16650} C_VEL
LIN {X 0,Y 289.595,Z 392.864,A -85,B 0,C 180,E1 -16651.391,E2 -16651.391} C_VEL
LIN {X 0,Y 289.55,Z 392.521,A -85,B 0,C 180,E1 -16652.782,E2 -16652.782} C_VEL
LIN {X 0,Y 289.521,Z 391.781,A -85,B 0,C 180,E1 -16654.176,E2 -16654.176} C_VEL
LIN {X 0,Y 289.477,Z 390.642,A -85,B 0,C 180,E1 -16655.573,E2 -16655.573} C_VEL
LIN {X 0,Y 289.653,Z 388.11,A -85,B 0,C 180,E1 -16657.669,E2 -16657.669} C_VEL
LIN {X 0,Y 290.056,Z 384.584,A -85,B 0,C 180,E1 -16659.765,E2 -16659.765} C_VEL
LIN {X 0,Y 290.717,Z 379.981,A -85,B 0,C 180,E1 -16661.858,E2 -16661.858} C_VEL
LIN {X 0,Y 292.123,Z 373.074,A -85,B 0,C 180,E1 -16664.276,E2 -16664.276} C_VEL
LIN {X 0,Y 293.625,Z 365.59,A -85,B 0,C 180,E1 -16666.334,E2 -16666.334} C_VEL
LIN {X 0,Y 295.372,Z 356.355,A -85,B 0,C 180,E1 -16668.377,E2 -16668.377} C_VEL
LIN {X 0,Y 297.471,Z 345.736,A -85,B 0,C 180,E1 -16670.214,E2 -16670.214} C_VEL
LIN {X 0,Y 299.573,Z 334.994,A -85,B 0,C 180,E1 -16671.684,E2 -16671.684} C_VEL
LIN {X 0,Y 301.261,Z 324.692,A -85,B 0,C 180,E1 -16672.82,E2 -16672.82} C_VEL
LIN {X 0,Y 303.083,Z 312.471,A -85,B 0,C 180,E1 -16673.85,E2 -16673.85} C_VEL
LIN {X 0,Y 304.652,Z 299.098,A -85,B 0,C 180,E1 -16674.67,E2 -16674.67} C_VEL
LIN {X 0,Y 305.602,Z 286.943,A -85,B 0,C 180,E1 -16675.179,E2 -16675.179} C_VEL
LIN {X 0,Y 307.61,Z 228.504,A -85,B 0,C 180,E1 -16676.709,E2 -16676.709} C_VEL
LIN {X 0,Y 305.105,Z 209.128,A -85,B 0,C 180,E1 -16677.583,E2 -16677.583} C_VEL
LIN {X 0,Y 301.532,Z 189.288,A -85,B 0,C 180,E1 -16678.636,E2 -16678.636} C_VEL
LIN {X 0,Y 300.03,Z 183.283,A -85,B 0,C 180,E1 -16679.019,E2 -16679.019} C_VEL
LIN {X 0,Y 297.514,Z 177.177,A -85,B 0,C 180,E1 -16679.597,E2 -16679.597} C_VEL
LIN {X 0,Y 295.432,Z 167.395,A -85,B 0,C 180,E1 -16682.765,E2 -16682.765} C_VEL
LIN {X 0,Y 292.76,Z 157.054,A -85,B 0,C 180,E1 -16686.41,E2 -16686.41} C_VEL
LIN {X 0,Y 291.392,Z 152.195,A -85,B 0,C 180,E1 -16688.31,E2 -16688.31} C_VEL
LIN {X 0,Y 291.351,Z 152.199,A -85,B 0,C 180,E1 -16692.486,E2 -16692.486} C_VEL
LIN {X 0,Y 291.33,Z 152.197,A -85,B 0,C 180,E1 -16696.362,E2 -16696.362} C_VEL
LIN {X 0,Y 291.398,Z 152.185,A -85,B 0,C 180,E1 -16700.514,E2 -16700.514} C_VEL
LIN {X 0,Y 291.433,Z 152.183,A -85,B 0,C 180,E1 -16702.923,E2 -16702.923} C_VEL
LIN {X 0,Y 291.345,Z 152.191,A -85,B 0,C 180,E1 -16706.301,E2 -16706.301} C_VEL
LIN {X 0,Y 291.386,Z 152.181,A -85,B 0,C 180,E1 -16710.26,E2 -16710.26} C_VEL
LIN {X 0,Y 291.415,Z 152.177,A -85,B 0,C 180,E1 -16714.271,E2 -16714.271} C_VEL
LIN {X 0,Y 291.373,Z 152.18,A -85,B 0,C 180,E1 -16717.299,E2 -16717.299} C_VEL
LIN {X 0,Y 291.457,Z 152.173,A -85,B 0,C 180,E1 -16720.27,E2 -16720.27} C_VEL
LIN {X 0,Y 291.554,Z 152.158,A -85,B 0,C 180,E1 -16724.623,E2 -16724.623} C_VEL
LIN {X 0,Y 291.536,Z 152.161,A -85,B 0,C 180,E1 -16728.88,E2 -16728.88} C_VEL
LIN {X 0,Y 291.708,Z 152.144,A -85,B 0,C 180,E1 -16731.688,E2 -16731.688} C_VEL
LIN {X 0,Y 291.629,Z 152.158,A -85,B 0,C 180,E1 -16734.468,E2 -16734.468} C_VEL
LIN {X 0,Y 291.888,Z 152.126,A -85,B 0,C 180,E1 -16738.62,E2 -16738.62} C_VEL
LIN {X 0,Y 291.888,Z 152.127,A -85,B 0,C 180,E1 -16741.379,E2 -16741.379} C_VEL
LIN {X 0,Y 291.733,Z 152.143,A -85,B 0,C 180,E1 -16746.918,E2 -16746.918} C_VEL
LIN {X 0,Y 291.573,Z 152.166,A -85,B 0,C 180,E1 -16749.713,E2 -16749.713} C_VEL
LIN {X 0,Y 291.52,Z 152.17,A -85,B 0,C 180,E1 -16753.95,E2 -16753.95} C_VEL
LIN {X 0,Y 291.485,Z 152.177,A -85,B 0,C 180,E1 -16756.818,E2 -16756.818} C_VEL
LIN {X 0,Y 291.455,Z 152.18,A -85,B 0,C 180,E1 -16759.878,E2 -16759.878} C_VEL
LIN {X 0,Y 291.427,Z 152.399,A -85,B 0,C 180,E1 -16762.416,E2 -16762.416} C_VEL
LIN {X 0,Y 291.583,Z 153.109,A -85,B 0,C 180,E1 -16762.684,E2 -16762.684} C_VEL
LIN {X 0,Y 293,Z 155.84,A -85,B 0,C 180,E1 -16762.986,E2 -16762.986} C_VEL
LIN {X 0,Y 299.75,Z 167.662,A -85,B 0,C 180,E1 -16764.312,E2 -16764.312} C_VEL
LIN {X 0,Y 305.44,Z 179.616,A -85,B 0,C 180,E1 -16765.421,E2 -16765.421} C_VEL
LIN {X 0,Y 308.979,Z 187.96,A -85,B 0,C 180,E1 -16766.099,E2 -16766.099} C_VEL
LIN {X 0,Y 306.285,Z 260.08,A -85,B 0,C 180,E1 -16767.99,E2 -16767.99} C_VEL
LIN {X 0,Y 305.358,Z 273.453,A -85,B 0,C 180,E1 -16768.609,E2 -16768.609} C_VEL
LIN {X 0,Y 304.185,Z 286.327,A -85,B 0,C 180,E1 -16769.499,E2 -16769.499} C_VEL
LIN {X 0,Y 302.752,Z 298.029,A -85,B 0,C 180,E1 -16770.591,E2 -16770.591} C_VEL
LIN {X 0,Y 301.182,Z 308.317,A -85,B 0,C 180,E1 -16771.806,E2 -16771.806} C_VEL
LIN {X 0,Y 299.444,Z 318.279,A -85,B 0,C 180,E1 -16773.268,E2 -16773.268} C_VEL
LIN {X 0,Y 297.661,Z 327.265,A -85,B 0,C 180,E1 -16774.896,E2 -16774.896} C_VEL
LIN {X 0,Y 295.823,Z 335.637,A -85,B 0,C 180,E1 -16776.775,E2 -16776.775} C_VEL
LIN {X 0,Y 294.214,Z 342.701,A -85,B 0,C 180,E1 -16778.749,E2 -16778.749} C_VEL
LIN {X 0,Y 292.709,Z 349.249,A -85,B 0,C 180,E1 -16781.075,E2 -16781.075} C_VEL
LIN {X 0,Y 291.436,Z 354.616,A -85,B 0,C 180,E1 -16783.66,E2 -16783.66} C_VEL
LIN {X 0,Y 290.749,Z 357.432,A -85,B 0,C 180,E1 -16785.494,E2 -16785.494} C_VEL
LIN {X 0,Y 290.188,Z 359.453,A -85,B 0,C 180,E1 -16787.303,E2 -16787.303} C_VEL
LIN {X 0,Y 289.839,Z 360.732,A -85,B 0,C 180,E1 -16789.104,E2 -16789.104} C_VEL
LIN {X 0,Y 289.597,Z 361.375,A -85,B 0,C 180,E1 -16790.948,E2 -16790.948} C_VEL
LIN {X 0,Y 289.449,Z 361.171,A -85,B 0,C 180,E1 -16793.25,E2 -16793.25} C_VEL
LIN {X 0,Y 289.588,Z 359.821,A -85,B 0,C 180,E1 -16795.603,E2 -16795.603} C_VEL
LIN {X 0,Y 289.909,Z 357.174,A -85,B 0,C 180,E1 -16798.046,E2 -16798.046} C_VEL
LIN {X 0,Y 290.481,Z 353.016,A -85,B 0,C 180,E1 -16800.574,E2 -16800.574} C_VEL
LIN {X 0,Y 291.072,Z 348.25,A -85,B 0,C 180,E1 -16802.693,E2 -16802.693} C_VEL
LIN {X 0,Y 292.092,Z 341.199,A -85,B 0,C 180,E1 -16805.098,E2 -16805.098} C_VEL
LIN {X 0,Y 293.138,Z 333.902,A -85,B 0,C 180,E1 -16807.071,E2 -16807.071} C_VEL
LIN {X 0,Y 294.447,Z 324.905,A -85,B 0,C 180,E1 -16809.021,E2 -16809.021} C_VEL
LIN {X 0,Y 295.825,Z 314.486,A -85,B 0,C 180,E1 -16810.826,E2 -16810.826} C_VEL
LIN {X 0,Y 297.123,Z 304.077,A -85,B 0,C 180,E1 -16812.27,E2 -16812.27} C_VEL
LIN {X 0,Y 298.403,Z 291.994,A -85,B 0,C 180,E1 -16813.583,E2 -16813.583} C_VEL
LIN {X 0,Y 299.402,Z 279.714,A -85,B 0,C 180,E1 -16814.61,E2 -16814.61} C_VEL
LIN {X 0,Y 300.229,Z 266.893,A -85,B 0,C 180,E1 -16815.382,E2 -16815.382} C_VEL
LIN {X 0,Y 300.773,Z 254.043,A -85,B 0,C 180,E1 -16815.884,E2 -16815.884} C_VEL
LIN {X 0,Y 302.842,Z 181.914,A -85,B 0,C 180,E1 -16817.712,E2 -16817.712} C_VEL
LIN {X 0,Y 295.811,Z 162.524,A -85,B 0,C 180,E1 -16818.783,E2 -16818.783} C_VEL
LIN {X 0,Y 291.678,Z 152.824,A -85,B 0,C 180,E1 -16819.392,E2 -16819.392} C_VEL
LIN {X 0,Y 291.557,Z 152.172,A -85,B 0,C 180,E1 -16819.427,E2 -16819.427} C_VEL
LIN {X 0,Y 291.737,Z 152.147,A -85,B 0,C 180,E1 -16823.082,E2 -16823.082} C_VEL
LIN {X 0,Y 291.888,Z 152.124,A -85,B 0,C 180,E1 -16828.62,E2 -16828.62} C_VEL
LIN {X 0,Y 291.888,Z 152.129,A -85,B 0,C 180,E1 -16831.38,E2 -16831.38} C_VEL
LIN {X 0,Y 291.61,Z 152.162,A -85,B 0,C 180,E1 -16835.532,E2 -16835.532} C_VEL
LIN {X 0,Y 291.667,Z 152.155,A -85,B 0,C 180,E1 -16838.911,E2 -16838.911} C_VEL
LIN {X 0,Y 291.516,Z 152.172,A -85,B 0,C 180,E1 -16842.531,E2 -16842.531} C_VEL
LIN {X 0,Y 291.506,Z 152.173,A -85,B 0,C 180,E1 -16845.379,E2 -16845.379} C_VEL
LIN {X 0,Y 291.423,Z 152.181,A -85,B 0,C 180,E1 -16849.86,E2 -16849.86} C_VEL
LIN {X 0,Y 291.382,Z 152.187,A -85,B 0,C 180,E1 -16854.207,E2 -16854.207} C_VEL
LIN {X 0,Y 291.425,Z 152.181,A -85,B 0,C 180,E1 -16857.271,E2 -16857.271} C_VEL
LIN {X 0,Y 291.337,Z 152.196,A -85,B 0,C 180,E1 -16860.437,E2 -16860.437} C_VEL
LIN {X 0,Y 291.344,Z 152.192,A -85,B 0,C 180,E1 -16863.698,E2 -16863.698} C_VEL
LIN {X 0,Y 291.375,Z 152.188,A -85,B 0,C 180,E1 -16867.254,E2 -16867.254} C_VEL
LIN {X 0,Y 291.331,Z 152.192,A -85,B 0,C 180,E1 -16870.643,E2 -16870.643} C_VEL
LIN {X 0,Y 291.289,Z 152.202,A -85,B 0,C 180,E1 -16874.402,E2 -16874.402} C_VEL
LIN {X 0,Y 291.325,Z 152.194,A -85,B 0,C 180,E1 -16878.404,E2 -16878.404} C_VEL
LIN {X 0,Y 291.362,Z 152.185,A -85,B 0,C 180,E1 -16881.16,E2 -16881.16} C_VEL
LIN {X 0,Y 291.361,Z 152.19,A -85,B 0,C 180,E1 -16884.626,E2 -16884.626} C_VEL
LIN {X 0,Y 291.371,Z 152.19,A -85,B 0,C 180,E1 -16887.951,E2 -16887.951} C_VEL
LIN {X 0,Y 291.38,Z 152.182,A -85,B 0,C 180,E1 -16891.158,E2 -16891.158} C_VEL
LIN {X 0,Y 291.434,Z 152.178,A -85,B 0,C 180,E1 -16893.061,E2 -16893.061} C_VEL
LIN {X 0,Y 290.795,Z 152.263,A -85,B 0,C 180,E1 -16894.214,E2 -16894.214} C_VEL
LIN {X 0,Y 287.89,Z 152.624,A -85,B 0,C 180,E1 -16896.09,E2 -16896.09} C_VEL
LIN {X 0,Y 285.421,Z 152.934,A -85,B 0,C 180,E1 -16897.613,E2 -16897.613} C_VEL
LIN {X 0,Y 284.395,Z 153.056,A -85,B 0,C 180,E1 -16898.795,E2 -16898.795} C_VEL
LIN {X 0,Y 284.331,Z 153.062,A -85,B 0,C 180,E1 -16899.196,E2 -16899.196} C_VEL
LIN {X 0,Y 284.424,Z 153.048,A -85,B 0,C 180,E1 -16902.752,E2 -16902.752} C_VEL
LIN {X 0,Y 284.481,Z 153.049,A -85,B 0,C 180,E1 -16905.697,E2 -16905.697} C_VEL
LIN {X 0,Y 284.566,Z 153.035,A -85,B 0,C 180,E1 -16910.045,E2 -16910.045} C_VEL
LIN {X 0,Y 284.697,Z 153.017,A -85,B 0,C 180,E1 -16912.91,E2 -16912.91} C_VEL
LIN {X 0,Y 284.855,Z 153,A -85,B 0,C 180,E1 -16918.587,E2 -16918.587} C_VEL
LIN {X 0,Y 284.855,Z 152.999,A -85,B 0,C 180,E1 -16921.414,E2 -16921.414} C_VEL
LIN {X 0,Y 284.693,Z 153.023,A -85,B 0,C 180,E1 -16927.09,E2 -16927.09} C_VEL
LIN {X 0,Y 284.566,Z 153.035,A -85,B 0,C 180,E1 -16929.956,E2 -16929.956} C_VEL
LIN {X 0,Y 284.481,Z 153.046,A -85,B 0,C 180,E1 -16934.303,E2 -16934.303} C_VEL
LIN {X 0,Y 284.425,Z 153.054,A -85,B 0,C 180,E1 -16937.249,E2 -16937.249} C_VEL
LIN {X 0,Y 284.377,Z 153.059,A -85,B 0,C 180,E1 -16940.243,E2 -16940.243} C_VEL
LIN {X 0,Y 284.338,Z 153.065,A -85,B 0,C 180,E1 -16944.847,E2 -16944.847} C_VEL
LIN {X 0,Y 284.332,Z 153.066,A -85,B 0,C 180,E1 -16948.011,E2 -16948.011} C_VEL
LIN {X 0,Y 284.296,Z 153.069,A -85,B 0,C 180,E1 -16951.275,E2 -16951.275} C_VEL
LIN {X 0,Y 284.362,Z 153.062,A -85,B 0,C 180,E1 -16955.354,E2 -16955.354} C_VEL
LIN {X 0,Y 284.333,Z 153.07,A -85,B 0,C 180,E1 -16958.166,E2 -16958.166} C_VEL
LIN {X 0,Y 284.302,Z 153.073,A -85,B 0,C 180,E1 -16961.871,E2 -16961.871} C_VEL
LIN {X 0,Y 284.275,Z 153.075,A -85,B 0,C 180,E1 -16966.193,E2 -16966.193} C_VEL
LIN {X 0,Y 284.353,Z 153.067,A -85,B 0,C 180,E1 -16970.013,E2 -16970.013} C_VEL
LIN {X 0,Y 284.354,Z 153.065,A -85,B 0,C 180,E1 -16973.618,E2 -16973.618} C_VEL
LIN {X 0,Y 284.377,Z 153.247,A -85,B 0,C 180,E1 -16975.272,E2 -16975.272} C_VEL
LIN {X 0,Y 287.013,Z 165.343,A -85,B 0,C 180,E1 -16979.055,E2 -16979.055} C_VEL
LIN {X 0,Y 289.115,Z 175.68,A -85,B 0,C 180,E1 -16982.143,E2 -16982.143} C_VEL
LIN {X 0,Y 288.834,Z 179.958,A -85,B 0,C 180,E1 -16983.313,E2 -16983.313} C_VEL
LIN {X 0,Y 293.876,Z 217.343,A -85,B 0,C 180,E1 -16984.772,E2 -16984.772} C_VEL
LIN {X 0,Y 295.157,Z 229.382,A -85,B 0,C 180,E1 -16985.202,E2 -16985.202} C_VEL
LIN {X 0,Y 293.433,Z 289.875,A -85,B 0,C 180,E1 -16986.816,E2 -16986.816} C_VEL
LIN {X 0,Y 292.539,Z 303.216,A -85,B 0,C 180,E1 -16987.441,E2 -16987.441} C_VEL
LIN {X 0,Y 291.289,Z 315.963,A -85,B 0,C 180,E1 -16988.319,E2 -16988.319} C_VEL
LIN {X 0,Y 289.911,Z 327.7,A -85,B 0,C 180,E1 -16989.42,E2 -16989.42} C_VEL
LIN {X 0,Y 288.376,Z 339.069,A -85,B 0,C 180,E1 -16990.792,E2 -16990.792} C_VEL
LIN {X 0,Y 286.952,Z 349.346,A -85,B 0,C 180,E1 -16992.357,E2 -16992.357} C_VEL
LIN {X 0,Y 285.675,Z 358.097,A -85,B 0,C 180,E1 -16994.007,E2 -16994.007} C_VEL
LIN {X 0,Y 284.504,Z 366.918,A -85,B 0,C 180,E1 -16996.063,E2 -16996.063} C_VEL
LIN {X 0,Y 283.465,Z 374.265,A -85,B 0,C 180,E1 -16998.197,E2 -16998.197} C_VEL
LIN {X 0,Y 282.977,Z 379.224,A -85,B 0,C 180,E1 -16999.988,E2 -16999.988} C_VEL
LIN {X 0,Y 282.627,Z 384.019,A -85,B 0,C 180,E1 -17002.139,E2 -17002.139} C_VEL
LIN {X 0,Y 282.524,Z 387.657,A -85,B 0,C 180,E1 -17004.289,E2 -17004.289} C_VEL
LIN {X 0,Y 282.487,Z 389.505,A -85,B 0,C 180,E1 -17005.72,E2 -17005.72} C_VEL
LIN {X 0,Y 282.506,Z 390.871,A -85,B 0,C 180,E1 -17007.148,E2 -17007.148} C_VEL
LIN {X 0,Y 282.551,Z 391.823,A -85,B 0,C 180,E1 -17008.575,E2 -17008.575} C_VEL
LIN {X 0,Y 282.631,Z 392.371,A -85,B 0,C 180,E1 -17010,E2 -17010} C_VEL
LIN {X 0,Y 282.508,Z 392.482,A -85,B 0,C 180,E1 -17011.425,E2 -17011.425} C_VEL
LIN {X 0,Y 282.474,Z 392.161,A -85,B 0,C 180,E1 -17012.852,E2 -17012.852} C_VEL
LIN {X 0,Y 282.371,Z 390.605,A -85,B 0,C 180,E1 -17015.391,E2 -17015.391} C_VEL
LIN {X 0,Y 282.491,Z 388.791,A -85,B 0,C 180,E1 -17017.146,E2 -17017.146} C_VEL
LIN {X 0,Y 282.855,Z 385.663,A -85,B 0,C 180,E1 -17019.294,E2 -17019.294} C_VEL
LIN {X 0,Y 283.452,Z 381.482,A -85,B 0,C 180,E1 -17021.441,E2 -17021.441} C_VEL
LIN {X 0,Y 284.739,Z 375.115,A -85,B 0,C 180,E1 -17023.925,E2 -17023.925} C_VEL
LIN {X 0,Y 286.175,Z 368.224,A -85,B 0,C 180,E1 -17026.038,E2 -17026.038} C_VEL
LIN {X 0,Y 287.994,Z 359.657,A -85,B 0,C 180,E1 -17028.147,E2 -17028.147} C_VEL
LIN {X 0,Y 289.783,Z 351.058,A -85,B 0,C 180,E1 -17029.848,E2 -17029.848} C_VEL
LIN {X 0,Y 292.041,Z 340.416,A -85,B 0,C 180,E1 -17031.53,E2 -17031.53} C_VEL
LIN {X 0,Y 293.987,Z 329.93,A -85,B 0,C 180,E1 -17032.859,E2 -17032.859} C_VEL
LIN {X 0,Y 295.939,Z 318.439,A -85,B 0,C 180,E1 -17033.997,E2 -17033.997} C_VEL
LIN {X 0,Y 297.698,Z 305.41,A -85,B 0,C 180,E1 -17034.96,E2 -17034.96} C_VEL
LIN {X 0,Y 299.022,Z 292.512,A -85,B 0,C 180,E1 -17035.633,E2 -17035.633} C_VEL
LIN {X 0,Y 299.749,Z 279.052,A -85,B 0,C 180,E1 -17036.079,E2 -17036.079} C_VEL
LIN {X 0,Y 301.506,Z 229.093,A -85,B 0,C 180,E1 -17037.397,E2 -17037.397} C_VEL
LIN {X 0,Y 299.049,Z 210.127,A -85,B 0,C 180,E1 -17038.294,E2 -17038.294} C_VEL
LIN {X 0,Y 295.853,Z 191.73,A -85,B 0,C 180,E1 -17039.299,E2 -17039.299} C_VEL
LIN {X 0,Y 294.498,Z 186.265,A -85,B 0,C 180,E1 -17039.66,E2 -17039.66} C_VEL
LIN {X 0,Y 290.258,Z 176.675,A -85,B 0,C 180,E1 -17040.615,E2 -17040.615} C_VEL
LIN {X 0,Y 288.051,Z 166.925,A -85,B 0,C 180,E1 -17043.947,E2 -17043.947} C_VEL
LIN {X 0,Y 286.352,Z 160.091,A -85,B 0,C 180,E1 -17046.445,E2 -17046.445} C_VEL
LIN {X 0,Y 284.345,Z 153.071,A -85,B 0,C 180,E1 -17049.298,E2 -17049.298} C_VEL
LIN {X 0,Y 284.3,Z 153.08,A -85,B 0,C 180,E1 -17052.131,E2 -17052.131} C_VEL
LIN {X 0,Y 284.274,Z 153.075,A -85,B 0,C 180,E1 -17056.192,E2 -17056.192} C_VEL
LIN {X 0,Y 284.352,Z 153.066,A -85,B 0,C 180,E1 -17060.013,E2 -17060.013} C_VEL
LIN {X 0,Y 284.355,Z 153.061,A -85,B 0,C 180,E1 -17063.617,E2 -17063.617} C_VEL
LIN {X 0,Y 284.308,Z 153.064,A -85,B 0,C 180,E1 -17067.189,E2 -17067.189} C_VEL
LIN {X 0,Y 284.358,Z 153.056,A -85,B 0,C 180,E1 -17070.376,E2 -17070.376} C_VEL
LIN {X 0,Y 284.377,Z 153.053,A -85,B 0,C 180,E1 -17073.586,E2 -17073.586} C_VEL
LIN {X 0,Y 284.332,Z 153.06,A -85,B 0,C 180,E1 -17076.704,E2 -17076.704} C_VEL
LIN {X 0,Y 284.402,Z 153.048,A -85,B 0,C 180,E1 -17081.261,E2 -17081.261} C_VEL
LIN {X 0,Y 284.491,Z 153.038,A -85,B 0,C 180,E1 -17084.459,E2 -17084.459} C_VEL
LIN {X 0,Y 284.487,Z 153.039,A -85,B 0,C 180,E1 -17088.601,E2 -17088.601} C_VEL
LIN {X 0,Y 284.658,Z 153.023,A -85,B 0,C 180,E1 -17091.481,E2 -17091.481} C_VEL
LIN {X 0,Y 284.6,Z 153.034,A -85,B 0,C 180,E1 -17094.331,E2 -17094.331} C_VEL
LIN {X 0,Y 284.854,Z 153.002,A -85,B 0,C 180,E1 -17098.586,E2 -17098.586} C_VEL
LIN {X 0,Y 284.854,Z 153.003,A -85,B 0,C 180,E1 -17101.413,E2 -17101.413} C_VEL
LIN {X 0,Y 284.685,Z 153.023,A -85,B 0,C 180,E1 -17107.09,E2 -17107.09} C_VEL
LIN {X 0,Y 284.517,Z 153.045,A -85,B 0,C 180,E1 -17109.957,E2 -17109.957} C_VEL
LIN {X 0,Y 284.48,Z 153.047,A -85,B 0,C 180,E1 -17114.303,E2 -17114.303} C_VEL
LIN {X 0,Y 284.424,Z 153.057,A -85,B 0,C 180,E1 -17117.248,E2 -17117.248} C_VEL
LIN {X 0,Y 284.361,Z 153.16,A -85,B 0,C 180,E1 -17121.427,E2 -17121.427} C_VEL
LIN {X 0,Y 284.462,Z 153.726,A -85,B 0,C 180,E1 -17121.609,E2 -17121.609} C_VEL
LIN {X 0,Y 285.745,Z 156.501,A -85,B 0,C 180,E1 -17121.91,E2 -17121.91} C_VEL
LIN {X 0,Y 287.028,Z 158.259,A -85,B 0,C 180,E1 -17122.171,E2 -17122.171} C_VEL
LIN {X 0,Y 293.252,Z 169.021,A -85,B 0,C 180,E1 -17123.468,E2 -17123.468} C_VEL
LIN {X 0,Y 299.187,Z 181.176,A -85,B 0,C 180,E1 -17124.67,E2 -17124.67} C_VEL
LIN {X 0,Y 303.003,Z 190.344,A -85,B 0,C 180,E1 -17125.45,E2 -17125.45} C_VEL
LIN {X 0,Y 300.174,Z 260.342,A -85,B 0,C 180,E1 -17127.316,E2 -17127.316} C_VEL
LIN {X 0,Y 299.195,Z 273.677,A -85,B 0,C 180,E1 -17127.939,E2 -17127.939} C_VEL
LIN {X 0,Y 298.044,Z 286.044,A -85,B 0,C 180,E1 -17128.799,E2 -17128.799} C_VEL
LIN {X 0,Y 296.411,Z 298.685,A -85,B 0,C 180,E1 -17129.993,E2 -17129.993} C_VEL
LIN {X 0,Y 294.767,Z 309.075,A -85,B 0,C 180,E1 -17131.252,E2 -17131.252} C_VEL
LIN {X 0,Y 292.797,Z 319.633,A -85,B 0,C 180,E1 -17132.85,E2 -17132.85} C_VEL
LIN {X 0,Y 290.698,Z 329.384,A -85,B 0,C 180,E1 -17134.716,E2 -17134.716} C_VEL
LIN {X 0,Y 288.628,Z 338.346,A -85,B 0,C 180,E1 -17136.878,E2 -17136.878} C_VEL
LIN {X 0,Y 286.848,Z 345.547,A -85,B 0,C 180,E1 -17139.114,E2 -17139.114} C_VEL
LIN {X 0,Y 285.275,Z 351.939,A -85,B 0,C 180,E1 -17141.695,E2 -17141.695} C_VEL
LIN {X 0,Y 284.129,Z 356.388,A -85,B 0,C 180,E1 -17144.167,E2 -17144.167} C_VEL
LIN {X 0,Y 283.49,Z 358.851,A -85,B 0,C 180,E1 -17146.041,E2 -17146.041} C_VEL
LIN {X 0,Y 282.919,Z 360.726,A -85,B 0,C 180,E1 -17148.179,E2 -17148.179} C_VEL
LIN {X 0,Y 282.552,Z 361.716,A -85,B 0,C 180,E1 -17150.45,E2 -17150.45} C_VEL
LIN {X 0,Y 282.402,Z 361.68,A -85,B 0,C 180,E1 -17152.784,E2 -17152.784} C_VEL
LIN {X 0,Y 282.458,Z 360.515,A -85,B 0,C 180,E1 -17155.194,E2 -17155.194} C_VEL
LIN {X 0,Y 282.754,Z 358.061,A -85,B 0,C 180,E1 -17157.681,E2 -17157.681} C_VEL
LIN {X 0,Y 283.306,Z 354.127,A -85,B 0,C 180,E1 -17160.255,E2 -17160.255} C_VEL
LIN {X 0,Y 283.913,Z 349.417,A -85,B 0,C 180,E1 -17162.501,E2 -17162.501} C_VEL
LIN {X 0,Y 284.852,Z 343.12,A -85,B 0,C 180,E1 -17164.812,E2 -17164.812} C_VEL
LIN {X 0,Y 285.885,Z 336.128,A -85,B 0,C 180,E1 -17166.838,E2 -17166.838} C_VEL
LIN {X 0,Y 287.212,Z 327.363,A -85,B 0,C 180,E1 -17168.881,E2 -17168.881} C_VEL
LIN {X 0,Y 288.518,Z 318.255,A -85,B 0,C 180,E1 -17170.599,E2 -17170.599} C_VEL
LIN {X 0,Y 289.878,Z 307.86,A -85,B 0,C 180,E1 -17172.176,E2 -17172.176} C_VEL
LIN {X 0,Y 291.305,Z 295.628,A -85,B 0,C 180,E1 -17173.641,E2 -17173.641} C_VEL
LIN {X 0,Y 292.357,Z 283.559,A -85,B 0,C 180,E1 -17174.756,E2 -17174.756} C_VEL
LIN {X 0,Y 293.368,Z 270.124,A -85,B 0,C 180,E1 -17175.653,E2 -17175.653} C_VEL
LIN {X 0,Y 293.986,Z 257.052,A -85,B 0,C 180,E1 -17176.242,E2 -17176.242} C_VEL
LIN {X 0,Y 296.087,Z 182.924,A -85,B 0,C 180,E1 -17178.187,E2 -17178.187} C_VEL
LIN {X 0,Y 289.56,Z 165.232,A -85,B 0,C 180,E1 -17179.203,E2 -17179.203} C_VEL
LIN {X 0,Y 284.738,Z 154.07,A -85,B 0,C 180,E1 -17179.93,E2 -17179.93} C_VEL
LIN {X 0,Y 284.536,Z 153.046,A -85,B 0,C 180,E1 -17180.003,E2 -17180.003} C_VEL
LIN {X 0,Y 284.688,Z 153.024,A -85,B 0,C 180,E1 -17182.91,E2 -17182.91} C_VEL
LIN {X 0,Y 284.854,Z 153.001,A -85,B 0,C 180,E1 -17188.586,E2 -17188.586} C_VEL
LIN {X 0,Y 284.854,Z 153.005,A -85,B 0,C 180,E1 -17191.414,E2 -17191.414} C_VEL
LIN {X 0,Y 284.579,Z 153.037,A -85,B 0,C 180,E1 -17195.669,E2 -17195.669} C_VEL
LIN {X 0,Y 284.609,Z 153.035,A -85,B 0,C 180,E1 -17198.982,E2 -17198.982} C_VEL
LIN {X 0,Y 284.472,Z 153.051,A -85,B 0,C 180,E1 -17202.847,E2 -17202.847} C_VEL
LIN {X 0,Y 284.422,Z 153.054,A -85,B 0,C 180,E1 -17205.772,E2 -17205.772} C_VEL
LIN {X 0,Y 284.367,Z 153.061,A -85,B 0,C 180,E1 -17210.243,E2 -17210.243} C_VEL
LIN {X 0,Y 284.339,Z 153.068,A -85,B 0,C 180,E1 -17214.846,E2 -17214.846} C_VEL
LIN {X 0,Y 284.334,Z 153.064,A -85,B 0,C 180,E1 -17218.01,E2 -17218.01} C_VEL
LIN {X 0,Y 284.295,Z 153.069,A -85,B 0,C 180,E1 -17221.274,E2 -17221.274} C_VEL
LIN {X 0,Y 284.34,Z 153.064,A -85,B 0,C 180,E1 -17225.348,E2 -17225.348} C_VEL
LIN {X 0,Y 284.311,Z 153.071,A -85,B 0,C 180,E1 -17228.169,E2 -17228.169} C_VEL
LIN {X 0,Y 284.268,Z 153.072,A -85,B 0,C 180,E1 -17232.124,E2 -17232.124} C_VEL
LIN {X 0,Y 284.254,Z 153.079,A -85,B 0,C 180,E1 -17236.189,E2 -17236.189} C_VEL
LIN {X 0,Y 284.306,Z 153.068,A -85,B 0,C 180,E1 -17240.024,E2 -17240.024} C_VEL
LIN {X 0,Y 284.335,Z 153.065,A -85,B 0,C 180,E1 -17243.615,E2 -17243.615} C_VEL
LIN {X 0,Y 284.307,Z 153.067,A -85,B 0,C 180,E1 -17247.19,E2 -17247.19} C_VEL
LIN {X 0,Y 284.357,Z 153.056,A -85,B 0,C 180,E1 -17250.376,E2 -17250.376} C_VEL
LIN {X 0,Y 284.376,Z 153.06,A -85,B 0,C 180,E1 -17253.587,E2 -17253.587} C_VEL
LIN {X 0,Y 284.332,Z 153.065,A -85,B 0,C 180,E1 -17256.704,E2 -17256.704} C_VEL
LIN {X 0,Y 284.331,Z 153.062,A -85,B 0,C 180,E1 -17259.196,E2 -17259.196} C_VEL
LIN {X 0,Y 283.737,Z 153.14,A -85,B 0,C 180,E1 -17260.378,E2 -17260.378} C_VEL
LIN {X 0,Y 280.981,Z 153.489,A -85,B 0,C 180,E1 -17262.306,E2 -17262.306} C_VEL
LIN {X 0,Y 278.587,Z 153.787,A -85,B 0,C 180,E1 -17263.871,E2 -17263.871} C_VEL
LIN {X 0,Y 277.525,Z 153.915,A -85,B 0,C 180,E1 -17265.082,E2 -17265.082} C_VEL
LIN {X 0,Y 277.422,Z 153.925,A -85,B 0,C 180,E1 -17265.493,E2 -17265.493} C_VEL
LIN {X 0,Y 277.506,Z 153.915,A -85,B 0,C 180,E1 -17269.789,E2 -17269.789} C_VEL
LIN {X 0,Y 277.652,Z 153.893,A -85,B 0,C 180,E1 -17272.729,E2 -17272.729} C_VEL
LIN {X 0,Y 277.821,Z 153.876,A -85,B 0,C 180,E1 -17278.551,E2 -17278.551} C_VEL
LIN {X 0,Y 277.821,Z 153.874,A -85,B 0,C 180,E1 -17281.45,E2 -17281.45} C_VEL
LIN {X 0,Y 277.648,Z 153.899,A -85,B 0,C 180,E1 -17287.271,E2 -17287.271} C_VEL
LIN {X 0,Y 277.506,Z 153.915,A -85,B 0,C 180,E1 -17290.212,E2 -17290.212} C_VEL
LIN {X 0,Y 277.434,Z 153.926,A -85,B 0,C 180,E1 -17294.674,E2 -17294.674} C_VEL
LIN {X 0,Y 277.345,Z 153.934,A -85,B 0,C 180,E1 -17299.234,E2 -17299.234} C_VEL
LIN {X 0,Y 277.292,Z 153.944,A -85,B 0,C 180,E1 -17304.158,E2 -17304.158} C_VEL
LIN {X 0,Y 277.326,Z 153.937,A -85,B 0,C 180,E1 -17307.506,E2 -17307.506} C_VEL
LIN {X 0,Y 277.272,Z 153.948,A -85,B 0,C 180,E1 -17310.482,E2 -17310.482} C_VEL
LIN {X 0,Y 277.255,Z 153.949,A -85,B 0,C 180,E1 -17313.895,E2 -17313.895} C_VEL
LIN {X 0,Y 277.288,Z 153.943,A -85,B 0,C 180,E1 -17317.467,E2 -17317.467} C_VEL
LIN {X 0,Y 277.24,Z 153.949,A -85,B 0,C 180,E1 -17321.231,E2 -17321.231} C_VEL
LIN {X 0,Y 277.213,Z 153.952,A -85,B 0,C 180,E1 -17325.225,E2 -17325.225} C_VEL
LIN {X 0,Y 277.263,Z 153.949,A -85,B 0,C 180,E1 -17329.503,E2 -17329.503} C_VEL
LIN {X 0,Y 277.289,Z 153.945,A -85,B 0,C 180,E1 -17332.534,E2 -17332.534} C_VEL
LIN {X 0,Y 277.321,Z 154.021,A -85,B 0,C 180,E1 -17334.793,E2 -17334.793} C_VEL
LIN {X 0,Y 279.886,Z 165.929,A -85,B 0,C 180,E1 -17338.622,E2 -17338.622} C_VEL
LIN {X 0,Y 282.007,Z 176.059,A -85,B 0,C 180,E1 -17341.738,E2 -17341.738} C_VEL
LIN {X 0,Y 282.039,Z 179.569,A -85,B 0,C 180,E1 -17342.743,E2 -17342.743} C_VEL
LIN {X 0,Y 286.821,Z 215.112,A -85,B 0,C 180,E1 -17344.185,E2 -17344.185} C_VEL
LIN {X 0,Y 288.495,Z 229.668,A -85,B 0,C 180,E1 -17344.732,E2 -17344.732} C_VEL
LIN {X 0,Y 286.751,Z 288.799,A -85,B 0,C 180,E1 -17346.338,E2 -17346.338} C_VEL
LIN {X 0,Y 285.804,Z 302.344,A -85,B 0,C 180,E1 -17346.975,E2 -17346.975} C_VEL
LIN {X 0,Y 284.552,Z 315.257,A -85,B 0,C 180,E1 -17347.874,E2 -17347.874} C_VEL
LIN {X 0,Y 283.025,Z 327.854,A -85,B 0,C 180,E1 -17349.087,E2 -17349.087} C_VEL
LIN {X 0,Y 281.454,Z 339.128,A -85,B 0,C 180,E1 -17350.49,E2 -17350.49} C_VEL
LIN {X 0,Y 279.991,Z 349.3,A -85,B 0,C 180,E1 -17352.092,E2 -17352.092} C_VEL
LIN {X 0,Y 278.616,Z 358.491,A -85,B 0,C 180,E1 -17353.891,E2 -17353.891} C_VEL
LIN {X 0,Y 277.376,Z 367.462,A -85,B 0,C 180,E1 -17356.072,E2 -17356.072} C_VEL
LIN {X 0,Y 276.312,Z 374.601,A -85,B 0,C 180,E1 -17358.259,E2 -17358.259} C_VEL
LIN {X 0,Y 275.79,Z 380.303,A -85,B 0,C 180,E1 -17360.466,E2 -17360.466} C_VEL
LIN {X 0,Y 275.495,Z 384.757,A -85,B 0,C 180,E1 -17362.672,E2 -17362.672} C_VEL
LIN {X 0,Y 275.443,Z 387.368,A -85,B 0,C 180,E1 -17364.327,E2 -17364.327} C_VEL
LIN {X 0,Y 275.409,Z 388.987,A -85,B 0,C 180,E1 -17365.609,E2 -17365.609} C_VEL
LIN {X 0,Y 275.431,Z 390.392,A -85,B 0,C 180,E1 -17367.075,E2 -17367.075} C_VEL
LIN {X 0,Y 275.464,Z 391.368,A -85,B 0,C 180,E1 -17368.538,E2 -17368.538} C_VEL
LIN {X 0,Y 275.542,Z 391.941,A -85,B 0,C 180,E1 -17370,E2 -17370} C_VEL
LIN {X 0,Y 275.424,Z 392.094,A -85,B 0,C 180,E1 -17371.462,E2 -17371.462} C_VEL
LIN {X 0,Y 275.398,Z 391.805,A -85,B 0,C 180,E1 -17372.926,E2 -17372.926} C_VEL
LIN {X 0,Y 275.282,Z 390.464,A -85,B 0,C 180,E1 -17375.326,E2 -17375.326} C_VEL
LIN {X 0,Y 275.419,Z 388.522,A -85,B 0,C 180,E1 -17377.33,E2 -17377.33} C_VEL
LIN {X 0,Y 275.816,Z 385.433,A -85,B 0,C 180,E1 -17379.533,E2 -17379.533} C_VEL
LIN {X 0,Y 276.447,Z 381.302,A -85,B 0,C 180,E1 -17381.735,E2 -17381.735} C_VEL
LIN {X 0,Y 277.833,Z 375.032,A -85,B 0,C 180,E1 -17384.278,E2 -17384.278} C_VEL
LIN {X 0,Y 279.355,Z 368.232,A -85,B 0,C 180,E1 -17386.441,E2 -17386.441} C_VEL
LIN {X 0,Y 281.195,Z 359.995,A -85,B 0,C 180,E1 -17388.544,E2 -17388.544} C_VEL
LIN {X 0,Y 283.135,Z 351.296,A -85,B 0,C 180,E1 -17390.335,E2 -17390.335} C_VEL
LIN {X 0,Y 285.475,Z 340.788,A -85,B 0,C 180,E1 -17392.051,E2 -17392.051} C_VEL
LIN {X 0,Y 287.746,Z 329.042,A -85,B 0,C 180,E1 -17393.575,E2 -17393.575} C_VEL
LIN {X 0,Y 289.808,Z 317.37,A -85,B 0,C 180,E1 -17394.728,E2 -17394.728} C_VEL
LIN {X 0,Y 291.623,Z 304.16,A -85,B 0,C 180,E1 -17395.708,E2 -17395.708} C_VEL
LIN {X 0,Y 293.015,Z 290.888,A -85,B 0,C 180,E1 -17396.389,E2 -17396.389} C_VEL
LIN {X 0,Y 293.894,Z 273.667,A -85,B 0,C 180,E1 -17396.927,E2 -17396.927} C_VEL
LIN {X 0,Y 295.497,Z 229.503,A -85,B 0,C 180,E1 -17398.128,E2 -17398.128} C_VEL
LIN {X 0,Y 292.948,Z 210.014,A -85,B 0,C 180,E1 -17399.093,E2 -17399.093} C_VEL
LIN {X 0,Y 289.854,Z 192.539,A -85,B 0,C 180,E1 -17400.097,E2 -17400.097} C_VEL
LIN {X 0,Y 288.857,Z 188.956,A -85,B 0,C 180,E1 -17400.362,E2 -17400.362} C_VEL
LIN {X 0,Y 284.487,Z 179.649,A -85,B 0,C 180,E1 -17401.341,E2 -17401.341} C_VEL
LIN {X 0,Y 282.974,Z 176.102,A -85,B 0,C 180,E1 -17401.747,E2 -17401.747} C_VEL
LIN {X 0,Y 281.235,Z 168.525,A -85,B 0,C 180,E1 -17404.445,E2 -17404.445} C_VEL
LIN {X 0,Y 279.46,Z 161.504,A -85,B 0,C 180,E1 -17407.125,E2 -17407.125} C_VEL
LIN {X 0,Y 277.282,Z 153.953,A -85,B 0,C 180,E1 -17410.283,E2 -17410.283} C_VEL
LIN {X 0,Y 277.229,Z 153.954,A -85,B 0,C 180,E1 -17413.194,E2 -17413.194} C_VEL
LIN {X 0,Y 277.237,Z 153.955,A -85,B 0,C 180,E1 -17417.32,E2 -17417.32} C_VEL
LIN {X 0,Y 277.267,Z 153.944,A -85,B 0,C 180,E1 -17420.677,E2 -17420.677} C_VEL
LIN {X 0,Y 277.305,Z 153.938,A -85,B 0,C 180,E1 -17424.344,E2 -17424.344} C_VEL
LIN {X 0,Y 277.244,Z 153.946,A -85,B 0,C 180,E1 -17427.836,E2 -17427.836} C_VEL
LIN {X 0,Y 277.271,Z 153.941,A -85,B 0,C 180,E1 -17431.21,E2 -17431.21} C_VEL
LIN {X 0,Y 277.309,Z 153.934,A -85,B 0,C 180,E1 -17434.479,E2 -17434.479} C_VEL
LIN {X 0,Y 277.268,Z 153.937,A -85,B 0,C 180,E1 -17437.653,E2 -17437.653} C_VEL
LIN {X 0,Y 277.344,Z 153.927,A -85,B 0,C 180,E1 -17440.766,E2 -17440.766} C_VEL
LIN {X 0,Y 277.434,Z 153.917,A -85,B 0,C 180,E1 -17445.325,E2 -17445.325} C_VEL
LIN {X 0,Y 277.506,Z 153.914,A -85,B 0,C 180,E1 -17449.788,E2 -17449.788} C_VEL
LIN {X 0,Y 277.652,Z 153.891,A -85,B 0,C 180,E1 -17452.729,E2 -17452.729} C_VEL
LIN {X 0,Y 277.82,Z 153.878,A -85,B 0,C 180,E1 -17458.55,E2 -17458.55} C_VEL
LIN {X 0,Y 277.82,Z 153.879,A -85,B 0,C 180,E1 -17461.449,E2 -17461.449} C_VEL
LIN {X 0,Y 277.639,Z 153.903,A -85,B 0,C 180,E1 -17467.271,E2 -17467.271} C_VEL
LIN {X 0,Y 277.46,Z 153.925,A -85,B 0,C 180,E1 -17470.213,E2 -17470.213} C_VEL
LIN {X 0,Y 277.433,Z 153.927,A -85,B 0,C 180,E1 -17474.674,E2 -17474.674} C_VEL
LIN {X 0,Y 277.344,Z 153.939,A -85,B 0,C 180,E1 -17479.234,E2 -17479.234} C_VEL
LIN {X 0,Y 277.363,Z 154.116,A -85,B 0,C 180,E1 -17480.429,E2 -17480.429} C_VEL
LIN {X 0,Y 278.472,Z 157.039,A -85,B 0,C 180,E1 -17480.739,E2 -17480.739} C_VEL
LIN {X 0,Y 279.937,Z 158.933,A -85,B 0,C 180,E1 -17481.058,E2 -17481.058} C_VEL
LIN {X 0,Y 286.799,Z 170.379,A -85,B 0,C 180,E1 -17482.56,E2 -17482.56} C_VEL
LIN {X 0,Y 293.413,Z 183.591,A -85,B 0,C 180,E1 -17483.973,E2 -17483.973} C_VEL
LIN {X 0,Y 297.058,Z 192.176,A -85,B 0,C 180,E1 -17484.743,E2 -17484.743} C_VEL
LIN {X 0,Y 294.147,Z 260.272,A -85,B 0,C 180,E1 -17486.588,E2 -17486.588} C_VEL
LIN {X 0,Y 293.141,Z 273.713,A -85,B 0,C 180,E1 -17487.224,E2 -17487.224} C_VEL
LIN {X 0,Y 291.977,Z 285.615,A -85,B 0,C 180,E1 -17488.056,E2 -17488.056} C_VEL
LIN {X 0,Y 290.443,Z 297.397,A -85,B 0,C 180,E1 -17489.157,E2 -17489.157} C_VEL
LIN {X 0,Y 288.682,Z 307.812,A -85,B 0,C 180,E1 -17490.394,E2 -17490.394} C_VEL
LIN {X 0,Y 286.608,Z 318.924,A -85,B 0,C 180,E1 -17492.065,E2 -17492.065} C_VEL
LIN {X 0,Y 284.593,Z 328.102,A -85,B 0,C 180,E1 -17493.789,E2 -17493.789} C_VEL
LIN {X 0,Y 282.804,Z 335.566,A -85,B 0,C 180,E1 -17495.513,E2 -17495.513} C_VEL
LIN {X 0,Y 281.033,Z 342.384,A -85,B 0,C 180,E1 -17497.441,E2 -17497.441} C_VEL
LIN {X 0,Y 279.263,Z 349.126,A -85,B 0,C 180,E1 -17499.865,E2 -17499.865} C_VEL
LIN {X 0,Y 278.111,Z 353.5,A -85,B 0,C 180,E1 -17501.885,E2 -17501.885} C_VEL
LIN {X 0,Y 277.164,Z 356.92,A -85,B 0,C 180,E1 -17503.918,E2 -17503.918} C_VEL
LIN {X 0,Y 276.216,Z 360.082,A -85,B 0,C 180,E1 -17506.609,E2 -17506.609} C_VEL
LIN {X 0,Y 275.759,Z 361.442,A -85,B 0,C 180,E1 -17508.499,E2 -17508.499} C_VEL
LIN {X 0,Y 275.496,Z 362.141,A -85,B 0,C 180,E1 -17510.376,E2 -17510.376} C_VEL
LIN {X 0,Y 275.33,Z 362.131,A -85,B 0,C 180,E1 -17512.307,E2 -17512.307} C_VEL
LIN {X 0,Y 275.327,Z 361.139,A -85,B 0,C 180,E1 -17514.769,E2 -17514.769} C_VEL
LIN {X 0,Y 275.656,Z 358.527,A -85,B 0,C 180,E1 -17517.629,E2 -17517.629} C_VEL
LIN {X 0,Y 276.111,Z 355.21,A -85,B 0,C 180,E1 -17519.93,E2 -17519.93} C_VEL
LIN {X 0,Y 276.646,Z 351.33,A -85,B 0,C 180,E1 -17521.954,E2 -17521.954} C_VEL
LIN {X 0,Y 277.593,Z 344.922,A -85,B 0,C 180,E1 -17524.507,E2 -17524.507} C_VEL
LIN {X 0,Y 278.641,Z 338.258,A -85,B 0,C 180,E1 -17526.594,E2 -17526.594} C_VEL
LIN {X 0,Y 280.022,Z 329.602,A -85,B 0,C 180,E1 -17528.759,E2 -17528.759} C_VEL
LIN {X 0,Y 281.449,Z 319.979,A -85,B 0,C 180,E1 -17530.679,E2 -17530.679} C_VEL
LIN {X 0,Y 282.808,Z 310.075,A -85,B 0,C 180,E1 -17532.277,E2 -17532.277} C_VEL
LIN {X 0,Y 284.114,Z 299.418,A -85,B 0,C 180,E1 -17533.658,E2 -17533.658} C_VEL
LIN {X 0,Y 285.424,Z 286.79,A -85,B 0,C 180,E1 -17534.925,E2 -17534.925} C_VEL
LIN {X 0,Y 286.277,Z 275.507,A -85,B 0,C 180,E1 -17535.789,E2 -17535.789} C_VEL
LIN {X 0,Y 287.076,Z 262.191,A -85,B 0,C 180,E1 -17536.507,E2 -17536.507} C_VEL
LIN {X 0,Y 287.734,Z 244.462,A -85,B 0,C 180,E1 -17537.055,E2 -17537.055} C_VEL
LIN {X 0,Y 289.401,Z 184.456,A -85,B 0,C 180,E1 -17538.655,E2 -17538.655} C_VEL
LIN {X 0,Y 283.641,Z 168.655,A -85,B 0,C 180,E1 -17539.589,E2 -17539.589} C_VEL
LIN {X 0,Y 277.628,Z 154.504,A -85,B 0,C 180,E1 -17540.529,E2 -17540.529} C_VEL
LIN {X 0,Y 277.532,Z 153.917,A -85,B 0,C 180,E1 -17540.602,E2 -17540.602} C_VEL
LIN {X 0,Y 277.643,Z 153.902,A -85,B 0,C 180,E1 -17542.729,E2 -17542.729} C_VEL
LIN {X 0,Y 277.82,Z 153.877,A -85,B 0,C 180,E1 -17548.551,E2 -17548.551} C_VEL
LIN {X 0,Y 277.82,Z 153.881,A -85,B 0,C 180,E1 -17551.45,E2 -17551.45} C_VEL
LIN {X 0,Y 277.604,Z 153.908,A -85,B 0,C 180,E1 -17557.272,E2 -17557.272} C_VEL
LIN {X 0,Y 277.457,Z 153.922,A -85,B 0,C 180,E1 -17560.213,E2 -17560.213} C_VEL
LIN {X 0,Y 277.409,Z 153.93,A -85,B 0,C 180,E1 -17564.675,E2 -17564.675} C_VEL
LIN {X 0,Y 277.317,Z 153.941,A -85,B 0,C 180,E1 -17569.236,E2 -17569.236} C_VEL
LIN {X 0,Y 277.297,Z 153.941,A -85,B 0,C 180,E1 -17573.923,E2 -17573.923} C_VEL
LIN {X 0,Y 277.327,Z 153.937,A -85,B 0,C 180,E1 -17577.506,E2 -17577.506} C_VEL
LIN {X 0,Y 277.271,Z 153.948,A -85,B 0,C 180,E1 -17580.481,E2 -17580.481} C_VEL
LIN {X 0,Y 277.246,Z 153.948,A -85,B 0,C 180,E1 -17583.896,E2 -17583.896} C_VEL
LIN {X 0,Y 277.266,Z 153.945,A -85,B 0,C 180,E1 -17587.469,E2 -17587.469} C_VEL
LIN {X 0,Y 277.208,Z 153.948,A -85,B 0,C 180,E1 -17591.237,E2 -17591.237} C_VEL
LIN {X 0,Y 277.2,Z 153.953,A -85,B 0,C 180,E1 -17595.226,E2 -17595.226} C_VEL
LIN {X 0,Y 277.221,Z 153.948,A -85,B 0,C 180,E1 -17599.512,E2 -17599.512} C_VEL
LIN {X 0,Y 277.272,Z 153.944,A -85,B 0,C 180,E1 -17602.532,E2 -17602.532} C_VEL
LIN {X 0,Y 277.246,Z 153.95,A -85,B 0,C 180,E1 -17606.104,E2 -17606.104} C_VEL
LIN {X 0,Y 277.26,Z 153.945,A -85,B 0,C 180,E1 -17609.539,E2 -17609.539} C_VEL
LIN {X 0,Y 277.358,Z 153.931,A -85,B 0,C 180,E1 -17612.864,E2 -17612.864} C_VEL
LIN {X 0,Y 277.296,Z 153.943,A -85,B 0,C 180,E1 -17616.077,E2 -17616.077} C_VEL
LIN {X 0,Y 277.344,Z 153.931,A -85,B 0,C 180,E1 -17620.766,E2 -17620.766} C_VEL
LIN {X 0,Y 277.434,Z 153.925,A -85,B 0,C 180,E1 -17625.326,E2 -17625.326} C_VEL
LIN {X 0,Y 277.422,Z 153.925,A -85,B 0,C 180,E1 -17625.493,E2 -17625.493} C_VEL
LIN {X 0,Y 276.725,Z 154.013,A -85,B 0,C 180,E1 -17626.705,E2 -17626.705} C_VEL
LIN {X 0,Y 273.929,Z 154.361,A -85,B 0,C 180,E1 -17628.683,E2 -17628.683} C_VEL
LIN {X 0,Y 271.605,Z 154.649,A -85,B 0,C 180,E1 -17630.289,E2 -17630.289} C_VEL
LIN {X 0,Y 270.639,Z 154.768,A -85,B 0,C 180,E1 -17631.533,E2 -17631.533} C_VEL
LIN {X 0,Y 270.575,Z 154.773,A -85,B 0,C 180,E1 -17631.953,E2 -17631.953} C_VEL
LIN {X 0,Y 270.421,Z 154.797,A -85,B 0,C 180,E1 -17635.529,E2 -17635.529} C_VEL
LIN {X 0,Y 270.787,Z 154.752,A -85,B 0,C 180,E1 -17638.513,E2 -17638.513} C_VEL
LIN {X 0,Y 270.787,Z 154.75,A -85,B 0,C 180,E1 -17641.488,E2 -17641.488} C_VEL
LIN {X 0,Y 270.607,Z 154.775,A -85,B 0,C 180,E1 -17647.462,E2 -17647.462} C_VEL
LIN {X 0,Y 270.441,Z 154.796,A -85,B 0,C 180,E1 -17650.481,E2 -17650.481} C_VEL
LIN {X 0,Y 270.403,Z 154.802,A -85,B 0,C 180,E1 -17655.065,E2 -17655.065} C_VEL
LIN {X 0,Y 270.301,Z 154.81,A -85,B 0,C 180,E1 -17659.756,E2 -17659.756} C_VEL
LIN {X 0,Y 270.238,Z 154.823,A -85,B 0,C 180,E1 -17664.589,E2 -17664.589} C_VEL
LIN {X 0,Y 270.272,Z 154.816,A -85,B 0,C 180,E1 -17667.909,E2 -17667.909} C_VEL
LIN {X 0,Y 270.185,Z 154.827,A -85,B 0,C 180,E1 -17671.349,E2 -17671.349} C_VEL
LIN {X 0,Y 270.216,Z 154.825,A -85,B 0,C 180,E1 -17674.904,E2 -17674.904} C_VEL
LIN {X 0,Y 270.223,Z 154.823,A -85,B 0,C 180,E1 -17678.717,E2 -17678.717} C_VEL
LIN {X 0,Y 270.193,Z 154.828,A -85,B 0,C 180,E1 -17682.555,E2 -17682.555} C_VEL
LIN {X 0,Y 270.183,Z 154.828,A -85,B 0,C 180,E1 -17686.748,E2 -17686.748} C_VEL
LIN {X 0,Y 270.214,Z 154.827,A -85,B 0,C 180,E1 -17689.442,E2 -17689.442} C_VEL
LIN {X 0,Y 270.258,Z 154.82,A -85,B 0,C 180,E1 -17693.722,E2 -17693.722} C_VEL
LIN {X 0,Y 270.289,Z 154.995,A -85,B 0,C 180,E1 -17694.366,E2 -17694.366} C_VEL
LIN {X 0,Y 272.969,Z 167.403,A -85,B 0,C 180,E1 -17698.462,E2 -17698.462} C_VEL
LIN {X 0,Y 275.145,Z 178.02,A -85,B 0,C 180,E1 -17701.801,E2 -17701.801} C_VEL
LIN {X 0,Y 275.235,Z 179.164,A -85,B 0,C 180,E1 -17702.143,E2 -17702.143} C_VEL
LIN {X 0,Y 280.004,Z 214.355,A -85,B 0,C 180,E1 -17703.629,E2 -17703.629} C_VEL
LIN {X 0,Y 281.812,Z 230.579,A -85,B 0,C 180,E1 -17704.255,E2 -17704.255} C_VEL
LIN {X 0,Y 280.04,Z 288.822,A -85,B 0,C 180,E1 -17705.883,E2 -17705.883} C_VEL
LIN {X 0,Y 278.996,Z 302.972,A -85,B 0,C 180,E1 -17706.576,E2 -17706.576} C_VEL
LIN {X 0,Y 277.713,Z 315.548,A -85,B 0,C 180,E1 -17707.495,E2 -17707.495} C_VEL
LIN {X 0,Y 276.15,Z 328.008,A -85,B 0,C 180,E1 -17708.736,E2 -17708.736} C_VEL
LIN {X 0,Y 274.539,Z 339.181,A -85,B 0,C 180,E1 -17710.173,E2 -17710.173} C_VEL
LIN {X 0,Y 273.192,Z 348.256,A -85,B 0,C 180,E1 -17711.631,E2 -17711.631} C_VEL
LIN {X 0,Y 271.677,Z 357.554,A -85,B 0,C 180,E1 -17713.468,E2 -17713.468} C_VEL
LIN {X 0,Y 270.573,Z 365.24,A -85,B 0,C 180,E1 -17715.33,E2 -17715.33} C_VEL
LIN {X 0,Y 269.514,Z 372.759,A -85,B 0,C 180,E1 -17717.577,E2 -17717.577} C_VEL
LIN {X 0,Y 268.896,Z 377.854,A -85,B 0,C 180,E1 -17719.458,E2 -17719.458} C_VEL
LIN {X 0,Y 268.497,Z 382.78,A -85,B 0,C 180,E1 -17721.723,E2 -17721.723} C_VEL
LIN {X 0,Y 268.354,Z 387.104,A -85,B 0,C 180,E1 -17724.384,E2 -17724.384} C_VEL
LIN {X 0,Y 268.358,Z 389.913,A -85,B 0,C 180,E1 -17726.998,E2 -17726.998} C_VEL
LIN {X 0,Y 268.381,Z 390.914,A -85,B 0,C 180,E1 -17728.499,E2 -17728.499} C_VEL
LIN {X 0,Y 268.453,Z 391.511,A -85,B 0,C 180,E1 -17730,E2 -17730} C_VEL
LIN {X 0,Y 268.343,Z 391.695,A -85,B 0,C 180,E1 -17731.501,E2 -17731.501} C_VEL
LIN {X 0,Y 268.321,Z 391.448,A -85,B 0,C 180,E1 -17733.003,E2 -17733.003} C_VEL
LIN {X 0,Y 268.22,Z 389.706,A -85,B 0,C 180,E1 -17736.016,E2 -17736.016} C_VEL
LIN {X 0,Y 268.34,Z 388.244,A -85,B 0,C 180,E1 -17737.525,E2 -17737.525} C_VEL
LIN {X 0,Y 268.765,Z 385.21,A -85,B 0,C 180,E1 -17739.786,E2 -17739.786} C_VEL
LIN {X 0,Y 269.456,Z 381.148,A -85,B 0,C 180,E1 -17742.044,E2 -17742.044} C_VEL
LIN {X 0,Y 270.947,Z 374.976,A -85,B 0,C 180,E1 -17744.649,E2 -17744.649} C_VEL
LIN {X 0,Y 272.539,Z 368.305,A -85,B 0,C 180,E1 -17746.847,E2 -17746.847} C_VEL
LIN {X 0,Y 274.465,Z 360.091,A -85,B 0,C 180,E1 -17749.016,E2 -17749.016} C_VEL
LIN {X 0,Y 276.482,Z 351.497,A -85,B 0,C 180,E1 -17750.847,E2 -17750.847} C_VEL
LIN {X 0,Y 278.922,Z 341.192,A -85,B 0,C 180,E1 -17752.597,E2 -17752.597} C_VEL
LIN {X 0,Y 281.292,Z 329.658,A -85,B 0,C 180,E1 -17754.15,E2 -17754.15} C_VEL
LIN {X 0,Y 283.425,Z 318.372,A -85,B 0,C 180,E1 -17755.324,E2 -17755.324} C_VEL
LIN {X 0,Y 285.141,Z 306.957,A -85,B 0,C 180,E1 -17756.239,E2 -17756.239} C_VEL
LIN {X 0,Y 286.748,Z 293.286,A -85,B 0,C 180,E1 -17757.012,E2 -17757.012} C_VEL
LIN {X 0,Y 287.631,Z 279.739,A -85,B 0,C 180,E1 -17757.513,E2 -17757.513} C_VEL
LIN {X 0,Y 289.604,Z 230.776,A -85,B 0,C 180,E1 -17758.856,E2 -17758.856} C_VEL
LIN {X 0,Y 287.134,Z 211.615,A -85,B 0,C 180,E1 -17759.837,E2 -17759.837} C_VEL
LIN {X 0,Y 284.256,Z 194.821,A -85,B 0,C 180,E1 -17760.844,E2 -17760.844} C_VEL
LIN {X 0,Y 283.591,Z 192.405,A -85,B 0,C 180,E1 -17761.03,E2 -17761.03} C_VEL
LIN {X 0,Y 279.22,Z 183.031,A -85,B 0,C 180,E1 -17762.05,E2 -17762.05} C_VEL
LIN {X 0,Y 275.759,Z 175.541,A -85,B 0,C 180,E1 -17762.953,E2 -17762.953} C_VEL
LIN {X 0,Y 273.473,Z 165.945,A -85,B 0,C 180,E1 -17766.607,E2 -17766.607} C_VEL
LIN {X 0,Y 270.829,Z 156.932,A -85,B 0,C 180,E1 -17770.447,E2 -17770.447} C_VEL
LIN {X 0,Y 270.201,Z 154.832,A -85,B 0,C 180,E1 -17771.421,E2 -17771.421} C_VEL
LIN {X 0,Y 270.163,Z 154.833,A -85,B 0,C 180,E1 -17775.382,E2 -17775.382} C_VEL
LIN {X 0,Y 270.237,Z 154.825,A -85,B 0,C 180,E1 -17779.445,E2 -17779.445} C_VEL
LIN {X 0,Y 270.257,Z 154.816,A -85,B 0,C 180,E1 -17783.721,E2 -17783.721} C_VEL
LIN {X 0,Y 270.204,Z 154.821,A -85,B 0,C 180,E1 -17786.892,E2 -17786.892} C_VEL
LIN {X 0,Y 270.197,Z 154.82,A -85,B 0,C 180,E1 -17790.382,E2 -17790.382} C_VEL
LIN {X 0,Y 270.261,Z 154.811,A -85,B 0,C 180,E1 -17793.763,E2 -17793.763} C_VEL
LIN {X 0,Y 270.21,Z 154.817,A -85,B 0,C 180,E1 -17797.036,E2 -17797.036} C_VEL
LIN {X 0,Y 270.3,Z 154.808,A -85,B 0,C 180,E1 -17800.244,E2 -17800.244} C_VEL
LIN {X 0,Y 270.402,Z 154.792,A -85,B 0,C 180,E1 -17804.935,E2 -17804.935} C_VEL
LIN {X 0,Y 270.441,Z 154.791,A -85,B 0,C 180,E1 -17809.519,E2 -17809.519} C_VEL
LIN {X 0,Y 270.61,Z 154.768,A -85,B 0,C 180,E1 -17812.538,E2 -17812.538} C_VEL
LIN {X 0,Y 270.786,Z 154.755,A -85,B 0,C 180,E1 -17818.512,E2 -17818.512} C_VEL
LIN {X 0,Y 270.786,Z 154.755,A -85,B 0,C 180,E1 -17821.487,E2 -17821.487} C_VEL
LIN {X 0,Y 270.597,Z 154.78,A -85,B 0,C 180,E1 -17827.461,E2 -17827.461} C_VEL
LIN {X 0,Y 270.411,Z 154.805,A -85,B 0,C 180,E1 -17830.482,E2 -17830.482} C_VEL
LIN {X 0,Y 270.401,Z 154.806,A -85,B 0,C 180,E1 -17835.064,E2 -17835.064} C_VEL
LIN {X 0,Y 270.312,Z 154.816,A -85,B 0,C 180,E1 -17839.162,E2 -17839.162} C_VEL
LIN {X 0,Y 271.29,Z 157.659,A -85,B 0,C 180,E1 -17839.483,E2 -17839.483} C_VEL
LIN {X 0,Y 273.018,Z 159.775,A -85,B 0,C 180,E1 -17839.882,E2 -17839.882} C_VEL
LIN {X 0,Y 275.053,Z 163.15,A -85,B 0,C 180,E1 -17840.377,E2 -17840.377} C_VEL
LIN {X 0,Y 282.062,Z 174.84,A -85,B 0,C 180,E1 -17841.983,E2 -17841.983} C_VEL
LIN {X 0,Y 288.424,Z 187.766,A -85,B 0,C 180,E1 -17843.405,E2 -17843.405} C_VEL
LIN {X 0,Y 291.106,Z 194.175,A -85,B 0,C 180,E1 -17844.008,E2 -17844.008} C_VEL
LIN {X 0,Y 288.123,Z 261.062,A -85,B 0,C 180,E1 -17845.86,E2 -17845.86} C_VEL
LIN {X 0,Y 287.005,Z 275.04,A -85,B 0,C 180,E1 -17846.544,E2 -17846.544} C_VEL
LIN {X 0,Y 285.693,Z 287.574,A -85,B 0,C 180,E1 -17847.467,E2 -17847.467} C_VEL
LIN {X 0,Y 283.925,Z 299.934,A -85,B 0,C 180,E1 -17848.696,E2 -17848.696} C_VEL
LIN {X 0,Y 282.023,Z 310.513,A -85,B 0,C 180,E1 -17850.038,E2 -17850.038} C_VEL
LIN {X 0,Y 279.836,Z 321.1,A -85,B 0,C 180,E1 -17851.737,E2 -17851.737} C_VEL
LIN {X 0,Y 277.493,Z 330.884,A -85,B 0,C 180,E1 -17853.716,E2 -17853.716} C_VEL
LIN {X 0,Y 275.452,Z 338.867,A -85,B 0,C 180,E1 -17855.738,E2 -17855.738} C_VEL
LIN {X 0,Y 273.431,Z 346.178,A -85,B 0,C 180,E1 -17858.088,E2 -17858.088} C_VEL
LIN {X 0,Y 271.618,Z 352.586,A -85,B 0,C 180,E1 -17860.781,E2 -17860.781} C_VEL
LIN {X 0,Y 270.376,Z 356.97,A -85,B 0,C 180,E1 -17863.297,E2 -17863.297} C_VEL
LIN {X 0,Y 269.575,Z 359.463,A -85,B 0,C 180,E1 -17865.259,E2 -17865.259} C_VEL
LIN {X 0,Y 268.98,Z 361.194,A -85,B 0,C 180,E1 -17867.209,E2 -17867.209} C_VEL
LIN {X 0,Y 268.511,Z 362.324,A -85,B 0,C 180,E1 -17869.38,E2 -17869.38} C_VEL
LIN {X 0,Y 268.259,Z 362.583,A -85,B 0,C 180,E1 -17871.809,E2 -17871.809} C_VEL
LIN {X 0,Y 268.245,Z 361.472,A -85,B 0,C 180,E1 -17874.803,E2 -17874.803} C_VEL
LIN {X 0,Y 268.444,Z 359.708,A -85,B 0,C 180,E1 -17876.906,E2 -17876.906} C_VEL
LIN {X 0,Y 268.967,Z 356.286,A -85,B 0,C 180,E1 -17879.573,E2 -17879.573} C_VEL
LIN {X 0,Y 269.579,Z 351.843,A -85,B 0,C 180,E1 -17882.014,E2 -17882.014} C_VEL
LIN {X 0,Y 270.517,Z 345.64,A -85,B 0,C 180,E1 -17884.568,E2 -17884.568} C_VEL
LIN {X 0,Y 271.608,Z 338.874,A -85,B 0,C 180,E1 -17886.759,E2 -17886.759} C_VEL
LIN {X 0,Y 272.95,Z 330.764,A -85,B 0,C 180,E1 -17888.871,E2 -17888.871} C_VEL
LIN {X 0,Y 274.472,Z 320.798,A -85,B 0,C 180,E1 -17890.933,E2 -17890.933} C_VEL
LIN {X 0,Y 276.089,Z 309.522,A -85,B 0,C 180,E1 -17892.787,E2 -17892.787} C_VEL
LIN {X 0,Y 277.494,Z 298.218,A -85,B 0,C 180,E1 -17894.24,E2 -17894.24} C_VEL
LIN {X 0,Y 278.784,Z 285.703,A -85,B 0,C 180,E1 -17895.492,E2 -17895.492} C_VEL
LIN {X 0,Y 279.775,Z 273.369,A -85,B 0,C 180,E1 -17896.402,E2 -17896.402} C_VEL
LIN {X 0,Y 280.5,Z 259.434,A -85,B 0,C 180,E1 -17897.105,E2 -17897.105} C_VEL
LIN {X 0,Y 282.885,Z 186.274,A -85,B 0,C 180,E1 -17899.125,E2 -17899.125} C_VEL
LIN {X 0,Y 277.373,Z 171.206,A -85,B 0,C 180,E1 -17900.043,E2 -17900.043} C_VEL
LIN {X 0,Y 270.683,Z 155.398,A -85,B 0,C 180,E1 -17901.132,E2 -17901.132} C_VEL
LIN {X 0,Y 270.579,Z 154.785,A -85,B 0,C 180,E1 -17901.191,E2 -17901.191} C_VEL
LIN {X 0,Y 270.538,Z 154.786,A -85,B 0,C 180,E1 -17904.036,E2 -17904.036} C_VEL
LIN {X 0,Y 270.786,Z 154.753,A -85,B 0,C 180,E1 -17908.513,E2 -17908.513} C_VEL
LIN {X 0,Y 270.786,Z 154.757,A -85,B 0,C 180,E1 -17911.487,E2 -17911.487} C_VEL
LIN {X 0,Y 270.565,Z 154.783,A -85,B 0,C 180,E1 -17917.462,E2 -17917.462} C_VEL
LIN {X 0,Y 270.409,Z 154.801,A -85,B 0,C 180,E1 -17920.482,E2 -17920.482} C_VEL
LIN {X 0,Y 270.368,Z 154.808,A -85,B 0,C 180,E1 -17925.067,E2 -17925.067} C_VEL
LIN {X 0,Y 270.257,Z 154.818,A -85,B 0,C 180,E1 -17929.759,E2 -17929.759} C_VEL
LIN {X 0,Y 270.238,Z 154.823,A -85,B 0,C 180,E1 -17934.589,E2 -17934.589} C_VEL
LIN {X 0,Y 270.272,Z 154.816,A -85,B 0,C 180,E1 -17937.908,E2 -17937.908} C_VEL
LIN {X 0,Y 270.184,Z 154.827,A -85,B 0,C 180,E1 -17941.348,E2 -17941.348} C_VEL
LIN {X 0,Y 270.201,Z 154.826,A -85,B 0,C 180,E1 -17944.905,E2 -17944.905} C_VEL
LIN {X 0,Y 270.196,Z 154.826,A -85,B 0,C 180,E1 -17948.71,E2 -17948.71} C_VEL
LIN {X 0,Y 270.164,Z 154.828,A -85,B 0,C 180,E1 -17953.249,E2 -17953.249} C_VEL
LIN {X 0,Y 270.17,Z 154.828,A -85,B 0,C 180,E1 -17957.442,E2 -17957.442} C_VEL
LIN {X 0,Y 270.206,Z 154.82,A -85,B 0,C 180,E1 -17961.374,E2 -17961.374} C_VEL
LIN {X 0,Y 270.202,Z 154.825,A -85,B 0,C 180,E1 -17965.095,E2 -17965.095} C_VEL
LIN {X 0,Y 270.199,Z 154.822,A -85,B 0,C 180,E1 -17969.131,E2 -17969.131} C_VEL
LIN {X 0,Y 270.263,Z 154.816,A -85,B 0,C 180,E1 -17972.146,E2 -17972.146} C_VEL
LIN {X 0,Y 270.237,Z 154.823,A -85,B 0,C 180,E1 -17975.538,E2 -17975.538} C_VEL
LIN {X 0,Y 270.3,Z 154.809,A -85,B 0,C 180,E1 -17980.245,E2 -17980.245} C_VEL
LIN {X 0,Y 270.402,Z 154.798,A -85,B 0,C 180,E1 -17984.936,E2 -17984.936} C_VEL
LIN {X 0,Y 270.441,Z 154.797,A -85,B 0,C 180,E1 -17989.519,E2 -17989.519} C_VEL
LIN {X 0,Y 270.575,Z 154.773,A -85,B 0,C 180,E1 -17991.953,E2 -17991.953} C_VEL
LIN {X 0,Y 269.968,Z 154.85,A -85,B 0,C 180,E1 -17993.193,E2 -17993.193} C_VEL
LIN {X 0,Y 267.22,Z 155.199,A -85,B 0,C 180,E1 -17995.216,E2 -17995.216} C_VEL
LIN {X 0,Y 264.858,Z 155.496,A -85,B 0,C 180,E1 -17996.861,E2 -17996.861} C_VEL
LIN {X 0,Y 263.836,Z 155.619,A -85,B 0,C 180,E1 -17998.133,E2 -17998.133} C_VEL
LIN {X 0,Y 263.749,Z 155.627,A -85,B 0,C 180,E1 -17998.564,E2 -17998.564} C_VEL
LIN {X 0,Y 263.751,Z 155.625,A -85,B 0,C 180,E1 -18001.527,E2 -18001.527} C_VEL
LIN {X 0,Y 263.569,Z 155.651,A -85,B 0,C 180,E1 -18007.662,E2 -18007.662} C_VEL
LIN {X 0,Y 263.374,Z 155.677,A -85,B 0,C 180,E1 -18010.766,E2 -18010.766} C_VEL
LIN {X 0,Y 263.351,Z 155.679,A -85,B 0,C 180,E1 -18015.478,E2 -18015.478} C_VEL
LIN {X 0,Y 263.263,Z 155.689,A -85,B 0,C 180,E1 -18020.307,E2 -18020.307} C_VEL
LIN {X 0,Y 263.193,Z 155.697,A -85,B 0,C 180,E1 -18025.293,E2 -18025.293} C_VEL
LIN {X 0,Y 263.18,Z 155.703,A -85,B 0,C 180,E1 -18028.73,E2 -18028.73} C_VEL
LIN {X 0,Y 263.134,Z 155.708,A -85,B 0,C 180,E1 -18032.289,E2 -18032.289} C_VEL
LIN {X 0,Y 263.19,Z 155.702,A -85,B 0,C 180,E1 -18035.978,E2 -18035.978} C_VEL
LIN {X 0,Y 263.14,Z 155.707,A -85,B 0,C 180,E1 -18039.867,E2 -18039.867} C_VEL
LIN {X 0,Y 263.13,Z 155.711,A -85,B 0,C 180,E1 -18043.983,E2 -18043.983} C_VEL
LIN {X 0,Y 263.156,Z 155.705,A -85,B 0,C 180,E1 -18048.399,E2 -18048.399} C_VEL
LIN {X 0,Y 263.19,Z 155.704,A -85,B 0,C 180,E1 -18052.108,E2 -18052.108} C_VEL
LIN {X 0,Y 263.225,Z 155.701,A -85,B 0,C 180,E1 -18053.83,E2 -18053.83} C_VEL
LIN {X 0,Y 265.936,Z 168.248,A -85,B 0,C 180,E1 -18058.093,E2 -18058.093} C_VEL
LIN {X 0,Y 268.133,Z 179.008,A -85,B 0,C 180,E1 -18061.522,E2 -18061.522} C_VEL
LIN {X 0,Y 269.412,Z 184.782,A -85,B 0,C 180,E1 -18061.82,E2 -18061.82} C_VEL
LIN {X 0,Y 274.184,Z 221.436,A -85,B 0,C 180,E1 -18063.369,E2 -18063.369} C_VEL
LIN {X 0,Y 275.155,Z 231.385,A -85,B 0,C 180,E1 -18063.752,E2 -18063.752} C_VEL
LIN {X 0,Y 273.332,Z 288.833,A -85,B 0,C 180,E1 -18065.404,E2 -18065.404} C_VEL
LIN {X 0,Y 272.277,Z 302.858,A -85,B 0,C 180,E1 -18066.114,E2 -18066.114} C_VEL
LIN {X 0,Y 270.974,Z 314.837,A -85,B 0,C 180,E1 -18067.004,E2 -18067.004} C_VEL
LIN {X 0,Y 269.512,Z 326.577,A -85,B 0,C 180,E1 -18068.186,E2 -18068.186} C_VEL
LIN {X 0,Y 267.892,Z 337.955,A -85,B 0,C 180,E1 -18069.659,E2 -18069.659} C_VEL
LIN {X 0,Y 266.386,Z 347.165,A -85,B 0,C 180,E1 -18071.144,E2 -18071.144} C_VEL
LIN {X 0,Y 264.753,Z 356.617,A -85,B 0,C 180,E1 -18073.022,E2 -18073.022} C_VEL
LIN {X 0,Y 263.915,Z 362.971,A -85,B 0,C 180,E1 -18074.556,E2 -18074.556} C_VEL
LIN {X 0,Y 262.711,Z 370.868,A -85,B 0,C 180,E1 -18076.857,E2 -18076.857} C_VEL
LIN {X 0,Y 261.874,Z 377.169,A -85,B 0,C 180,E1 -18079.172,E2 -18079.172} C_VEL
LIN {X 0,Y 261.436,Z 382.159,A -85,B 0,C 180,E1 -18081.497,E2 -18081.497} C_VEL
LIN {X 0,Y 261.26,Z 385.973,A -85,B 0,C 180,E1 -18083.823,E2 -18083.823} C_VEL
LIN {X 0,Y 261.244,Z 387.923,A -85,B 0,C 180,E1 -18085.371,E2 -18085.371} C_VEL
LIN {X 0,Y 261.287,Z 389.429,A -85,B 0,C 180,E1 -18086.916,E2 -18086.916} C_VEL
LIN {X 0,Y 261.3,Z 390.458,A -85,B 0,C 180,E1 -18088.459,E2 -18088.459} C_VEL
LIN {X 0,Y 261.367,Z 391.08,A -85,B 0,C 180,E1 -18090,E2 -18090} C_VEL
LIN {X 0,Y 261.263,Z 391.289,A -85,B 0,C 180,E1 -18091.541,E2 -18091.541} C_VEL
LIN {X 0,Y 261.223,Z 391.091,A -85,B 0,C 180,E1 -18093.084,E2 -18093.084} C_VEL
LIN {X 0,Y 261.144,Z 389.409,A -85,B 0,C 180,E1 -18096.18,E2 -18096.18} C_VEL
LIN {X 0,Y 261.286,Z 387.974,A -85,B 0,C 180,E1 -18097.729,E2 -18097.729} C_VEL
LIN {X 0,Y 261.724,Z 384.996,A -85,B 0,C 180,E1 -18100.052,E2 -18100.052} C_VEL
LIN {X 0,Y 262.479,Z 380.993,A -85,B 0,C 180,E1 -18102.369,E2 -18102.369} C_VEL
LIN {X 0,Y 263.797,Z 375.873,A -85,B 0,C 180,E1 -18104.661,E2 -18104.661} C_VEL
LIN {X 0,Y 265.721,Z 368.447,A -85,B 0,C 180,E1 -18107.255,E2 -18107.255} C_VEL
LIN {X 0,Y 267.796,Z 360.083,A -85,B 0,C 180,E1 -18109.549,E2 -18109.549} C_VEL
LIN {X 0,Y 269.87,Z 351.776,A -85,B 0,C 180,E1 -18111.382,E2 -18111.382} C_VEL
LIN {X 0,Y 272.401,Z 341.682,A -85,B 0,C 180,E1 -18113.169,E2 -18113.169} C_VEL
LIN {X 0,Y 274.872,Z 330.339,A -85,B 0,C 180,E1 -18114.751,E2 -18114.751} C_VEL
LIN {X 0,Y 277.072,Z 319.304,A -85,B 0,C 180,E1 -18115.947,E2 -18115.947} C_VEL
LIN {X 0,Y 279.005,Z 307.201,A -85,B 0,C 180,E1 -18116.962,E2 -18116.962} C_VEL
LIN {X 0,Y 280.694,Z 293.822,A -85,B 0,C 180,E1 -18117.745,E2 -18117.745} C_VEL
LIN {X 0,Y 281.603,Z 280.915,A -85,B 0,C 180,E1 -18118.255,E2 -18118.255} C_VEL
LIN {X 0,Y 283.711,Z 231.831,A -85,B 0,C 180,E1 -18119.636,E2 -18119.636} C_VEL
LIN {X 0,Y 281.349,Z 212.652,A -85,B 0,C 180,E1 -18120.656,E2 -18120.656} C_VEL
LIN {X 0,Y 278.586,Z 196.399,A -85,B 0,C 180,E1 -18121.668,E2 -18121.668} C_VEL
LIN {X 0,Y 273.025,Z 184.25,A -85,B 0,C 180,E1 -18123.049,E2 -18123.049} C_VEL
LIN {X 0,Y 270.109,Z 178.547,A -85,B 0,C 180,E1 -18123.791,E2 -18123.791} C_VEL
LIN {X 0,Y 268.431,Z 174.983,A -85,B 0,C 180,E1 -18124.284,E2 -18124.284} C_VEL
LIN {X 0,Y 266.592,Z 167.409,A -85,B 0,C 180,E1 -18127.325,E2 -18127.325} C_VEL
LIN {X 0,Y 264.361,Z 159.682,A -85,B 0,C 180,E1 -18130.74,E2 -18130.74} C_VEL
LIN {X 0,Y 263.155,Z 155.71,A -85,B 0,C 180,E1 -18132.685,E2 -18132.685} C_VEL
LIN {X 0,Y 263.132,Z 155.709,A -85,B 0,C 180,E1 -18136.149,E2 -18136.149} C_VEL
LIN {X 0,Y 263.155,Z 155.705,A -85,B 0,C 180,E1 -18140.136,E2 -18140.136} C_VEL
LIN {X 0,Y 263.19,Z 155.695,A -85,B 0,C 180,E1 -18144.022,E2 -18144.022} C_VEL
LIN {X 0,Y 263.133,Z 155.703,A -85,B 0,C 180,E1 -18147.711,E2 -18147.711} C_VEL
LIN {X 0,Y 263.196,Z 155.699,A -85,B 0,C 180,E1 -18151.785,E2 -18151.785} C_VEL
LIN {X 0,Y 263.201,Z 155.695,A -85,B 0,C 180,E1 -18155.212,E2 -18155.212} C_VEL
LIN {X 0,Y 263.262,Z 155.688,A -85,B 0,C 180,E1 -18159.693,E2 -18159.693} C_VEL
LIN {X 0,Y 263.35,Z 155.671,A -85,B 0,C 180,E1 -18164.522,E2 -18164.522} C_VEL
LIN {X 0,Y 263.373,Z 155.67,A -85,B 0,C 180,E1 -18169.234,E2 -18169.234} C_VEL
LIN {X 0,Y 263.572,Z 155.645,A -85,B 0,C 180,E1 -18172.338,E2 -18172.338} C_VEL
LIN {X 0,Y 263.75,Z 155.631,A -85,B 0,C 180,E1 -18178.473,E2 -18178.473} C_VEL
LIN {X 0,Y 263.75,Z 155.632,A -85,B 0,C 180,E1 -18181.527,E2 -18181.527} C_VEL
LIN {X 0,Y 263.557,Z 155.657,A -85,B 0,C 180,E1 -18187.662,E2 -18187.662} C_VEL
LIN {X 0,Y 263.354,Z 155.681,A -85,B 0,C 180,E1 -18190.766,E2 -18190.766} C_VEL
LIN {X 0,Y 263.349,Z 155.682,A -85,B 0,C 180,E1 -18195.478,E2 -18195.478} C_VEL
LIN {X 0,Y 263.262,Z 155.845,A -85,B 0,C 180,E1 -18197.828,E2 -18197.828} C_VEL
LIN {X 0,Y 264.293,Z 158.574,A -85,B 0,C 180,E1 -18198.157,E2 -18198.157} C_VEL
LIN {X 0,Y 266.153,Z 160.812,A -85,B 0,C 180,E1 -18198.623,E2 -18198.623} C_VEL
LIN {X 0,Y 268.238,Z 164.163,A -85,B 0,C 180,E1 -18199.166,E2 -18199.166} C_VEL
LIN {X 0,Y 275.748,Z 176.403,A -85,B 0,C 180,E1 -18201,E2 -18201} C_VEL
LIN {X 0,Y 281.493,Z 187.598,A -85,B 0,C 180,E1 -18202.349,E2 -18202.349} C_VEL
LIN {X 0,Y 285.215,Z 196.128,A -85,B 0,C 180,E1 -18203.219,E2 -18203.219} C_VEL
LIN {X 0,Y 282.191,Z 261.665,A -85,B 0,C 180,E1 -18205.093,E2 -18205.093} C_VEL
LIN {X 0,Y 281.082,Z 275.03,A -85,B 0,C 180,E1 -18205.76,E2 -18205.76} C_VEL
LIN {X 0,Y 279.821,Z 286.523,A -85,B 0,C 180,E1 -18206.597,E2 -18206.597} C_VEL
LIN {X 0,Y 278.043,Z 298.757,A -85,B 0,C 180,E1 -18207.788,E2 -18207.788} C_VEL
LIN {X 0,Y 276.097,Z 309.302,A -85,B 0,C 180,E1 -18209.106,E2 -18209.106} C_VEL
LIN {X 0,Y 273.953,Z 319.608,A -85,B 0,C 180,E1 -18210.727,E2 -18210.727} C_VEL
LIN {X 0,Y 271.843,Z 328.364,A -85,B 0,C 180,E1 -18212.429,E2 -18212.429} C_VEL
LIN {X 0,Y 269.571,Z 336.828,A -85,B 0,C 180,E1 -18214.472,E2 -18214.472} C_VEL
LIN {X 0,Y 267.556,Z 343.741,A -85,B 0,C 180,E1 -18216.551,E2 -18216.551} C_VEL
LIN {X 0,Y 265.898,Z 349.368,A -85,B 0,C 180,E1 -18218.664,E2 -18218.664} C_VEL
LIN {X 0,Y 264.541,Z 353.867,A -85,B 0,C 180,E1 -18220.788,E2 -18220.788} C_VEL
LIN {X 0,Y 263.496,Z 357.262,A -85,B 0,C 180,E1 -18222.821,E2 -18222.821} C_VEL
LIN {X 0,Y 262.956,Z 358.861,A -85,B 0,C 180,E1 -18224.019,E2 -18224.019} C_VEL
LIN {X 0,Y 262.12,Z 361.224,A -85,B 0,C 180,E1 -18226.379,E2 -18226.379} C_VEL
LIN {X 0,Y 261.562,Z 362.621,A -85,B 0,C 180,E1 -18228.793,E2 -18228.793} C_VEL
LIN {X 0,Y 261.172,Z 362.965,A -85,B 0,C 180,E1 -18231.763,E2 -18231.763} C_VEL
LIN {X 0,Y 261.139,Z 362.359,A -85,B 0,C 180,E1 -18233.841,E2 -18233.841} C_VEL
LIN {X 0,Y 261.297,Z 360.481,A -85,B 0,C 180,E1 -18236.49,E2 -18236.49} C_VEL
LIN {X 0,Y 261.812,Z 357.078,A -85,B 0,C 180,E1 -18239.335,E2 -18239.335} C_VEL
LIN {X 0,Y 262.493,Z 352.335,A -85,B 0,C 180,E1 -18242.072,E2 -18242.072} C_VEL
LIN {X 0,Y 263.485,Z 346.044,A -85,B 0,C 180,E1 -18244.737,E2 -18244.737} C_VEL
LIN {X 0,Y 264.58,Z 339.509,A -85,B 0,C 180,E1 -18246.916,E2 -18246.916} C_VEL
LIN {X 0,Y 265.971,Z 331.377,A -85,B 0,C 180,E1 -18249.101,E2 -18249.101} C_VEL
LIN {X 0,Y 267.428,Z 322.099,A -85,B 0,C 180,E1 -18251.098,E2 -18251.098} C_VEL
LIN {X 0,Y 268.985,Z 311.624,A -85,B 0,C 180,E1 -18252.906,E2 -18252.906} C_VEL
LIN {X 0,Y 270.481,Z 300.468,A -85,B 0,C 180,E1 -18254.441,E2 -18254.441} C_VEL
LIN {X 0,Y 271.905,Z 287.719,A -85,B 0,C 180,E1 -18255.786,E2 -18255.786} C_VEL
LIN {X 0,Y 272.877,Z 276.129,A -85,B 0,C 180,E1 -18256.713,E2 -18256.713} C_VEL
LIN {X 0,Y 273.697,Z 263.423,A -85,B 0,C 180,E1 -18257.436,E2 -18257.436} C_VEL
LIN {X 0,Y 274.325,Z 248.123,A -85,B 0,C 180,E1 -18257.952,E2 -18257.952} C_VEL
LIN {X 0,Y 276.29,Z 187.82,A -85,B 0,C 180,E1 -18259.628,E2 -18259.628} C_VEL
LIN {X 0,Y 271.146,Z 173.822,A -85,B 0,C 180,E1 -18260.507,E2 -18260.507} C_VEL
LIN {X 0,Y 263.636,Z 156.247,A -85,B 0,C 180,E1 -18261.766,E2 -18261.766} C_VEL
LIN {X 0,Y 263.54,Z 155.661,A -85,B 0,C 180,E1 -18261.807,E2 -18261.807} C_VEL
LIN {X 0,Y 263.376,Z 155.678,A -85,B 0,C 180,E1 -18265.409,E2 -18265.409} C_VEL
LIN {X 0,Y 263.75,Z 155.63,A -85,B 0,C 180,E1 -18268.473,E2 -18268.473} C_VEL
LIN {X 0,Y 263.75,Z 155.633,A -85,B 0,C 180,E1 -18271.527,E2 -18271.527} C_VEL
LIN {X 0,Y 263.528,Z 155.659,A -85,B 0,C 180,E1 -18277.663,E2 -18277.663} C_VEL
LIN {X 0,Y 263.349,Z 155.682,A -85,B 0,C 180,E1 -18280.767,E2 -18280.767} C_VEL
LIN {X 0,Y 263.31,Z 155.685,A -85,B 0,C 180,E1 -18285.48,E2 -18285.48} C_VEL
LIN {X 0,Y 263.237,Z 155.694,A -85,B 0,C 180,E1 -18290.309,E2 -18290.309} C_VEL
LIN {X 0,Y 263.193,Z 155.699,A -85,B 0,C 180,E1 -18295.293,E2 -18295.293} C_VEL
LIN {X 0,Y 263.18,Z 155.704,A -85,B 0,C 180,E1 -18298.729,E2 -18298.729} C_VEL
LIN {X 0,Y 263.132,Z 155.708,A -85,B 0,C 180,E1 -18302.288,E2 -18302.288} C_VEL
LIN {X 0,Y 263.162,Z 155.703,A -85,B 0,C 180,E1 -18305.982,E2 -18305.982} C_VEL
LIN {X 0,Y 263.104,Z 155.709,A -85,B 0,C 180,E1 -18309.872,E2 -18309.872} C_VEL
LIN {X 0,Y 263.121,Z 155.708,A -85,B 0,C 180,E1 -18313.984,E2 -18313.984} C_VEL
LIN {X 0,Y 263.123,Z 155.705,A -85,B 0,C 180,E1 -18318.407,E2 -18318.407} C_VEL
LIN {X 0,Y 263.193,Z 155.696,A -85,B 0,C 180,E1 -18323.233,E2 -18323.233} C_VEL
LIN {X 0,Y 263.166,Z 155.705,A -85,B 0,C 180,E1 -18325.888,E2 -18325.888} C_VEL
LIN {X 0,Y 263.14,Z 155.703,A -85,B 0,C 180,E1 -18329.506,E2 -18329.506} C_VEL
LIN {X 0,Y 263.19,Z 155.695,A -85,B 0,C 180,E1 -18333.003,E2 -18333.003} C_VEL
LIN {X 0,Y 263.154,Z 155.704,A -85,B 0,C 180,E1 -18336.385,E2 -18336.385} C_VEL
LIN {X 0,Y 263.262,Z 155.689,A -85,B 0,C 180,E1 -18339.694,E2 -18339.694} C_VEL
LIN {X 0,Y 263.35,Z 155.675,A -85,B 0,C 180,E1 -18344.522,E2 -18344.522} C_VEL
LIN {X 0,Y 263.373,Z 155.679,A -85,B 0,C 180,E1 -18349.235,E2 -18349.235} C_VEL
LIN {X 0,Y 263.572,Z 155.645,A -85,B 0,C 180,E1 -18352.339,E2 -18352.339} C_VEL
LIN {X 0,Y 263.749,Z 155.627,A -85,B 0,C 180,E1 -18358.564,E2 -18358.564} C_VEL
LIN {X 0,Y 263.022,Z 155.719,A -85,B 0,C 180,E1 -18359.838,E2 -18359.838} C_VEL
LIN {X 0,Y 259.984,Z 156.093,A -85,B 0,C 180,E1 -18361.909,E2 -18361.909} C_VEL
LIN {X 0,Y 257.454,Z 156.407,A -85,B 0,C 180,E1 -18363.594,E2 -18363.594} C_VEL
LIN {X 0,Y 256.426,Z 156.538,A -85,B 0,C 180,E1 -18364.906,E2 -18364.906} C_VEL
LIN {X 0,Y 256.373,Z 156.541,A -85,B 0,C 180,E1 -18365.35,E2 -18365.35} C_VEL
LIN {X 0,Y 256.537,Z 156.527,A -85,B 0,C 180,E1 -18367.873,E2 -18367.873} C_VEL
LIN {X 0,Y 256.31,Z 156.553,A -85,B 0,C 180,E1 -18371.066,E2 -18371.066} C_VEL
LIN {X 0,Y 256.3,Z 156.557,A -85,B 0,C 180,E1 -18375.915,E2 -18375.915} C_VEL
LIN {X 0,Y 256.163,Z 156.575,A -85,B 0,C 180,E1 -18380.896,E2 -18380.896} C_VEL
LIN {X 0,Y 256.171,Z 156.572,A -85,B 0,C 180,E1 -18385.13,E2 -18385.13} C_VEL
LIN {X 0,Y 256.114,Z 156.582,A -85,B 0,C 180,E1 -18389.6,E2 -18389.6} C_VEL
LIN {X 0,Y 256.086,Z 156.584,A -85,B 0,C 180,E1 -18393.291,E2 -18393.291} C_VEL
LIN {X 0,Y 256.141,Z 156.577,A -85,B 0,C 180,E1 -18397.279,E2 -18397.279} C_VEL
LIN {X 0,Y 256.086,Z 156.585,A -85,B 0,C 180,E1 -18401.198,E2 -18401.198} C_VEL
LIN {X 0,Y 256.064,Z 156.588,A -85,B 0,C 180,E1 -18405.529,E2 -18405.529} C_VEL
LIN {X 0,Y 256.086,Z 156.585,A -85,B 0,C 180,E1 -18408.803,E2 -18408.803} C_VEL
LIN {X 0,Y 256.191,Z 156.704,A -85,B 0,C 180,E1 -18413.369,E2 -18413.369} C_VEL
LIN {X 0,Y 258.666,Z 168.141,A -85,B 0,C 180,E1 -18417.382,E2 -18417.382} C_VEL
LIN {X 0,Y 260.85,Z 178.451,A -85,B 0,C 180,E1 -18420.828,E2 -18420.828} C_VEL
LIN {X 0,Y 262.702,Z 184.897,A -85,B 0,C 180,E1 -18421.214,E2 -18421.214} C_VEL
LIN {X 0,Y 267.51,Z 221.682,A -85,B 0,C 180,E1 -18422.828,E2 -18422.828} C_VEL
LIN {X 0,Y 268.545,Z 231.238,A -85,B 0,C 180,E1 -18423.215,E2 -18423.215} C_VEL
LIN {X 0,Y 266.672,Z 287.765,A -85,B 0,C 180,E1 -18424.872,E2 -18424.872} C_VEL
LIN {X 0,Y 265.623,Z 301.708,A -85,B 0,C 180,E1 -18425.581,E2 -18425.581} C_VEL
LIN {X 0,Y 264.281,Z 313.926,A -85,B 0,C 180,E1 -18426.491,E2 -18426.491} C_VEL
LIN {X 0,Y 262.667,Z 326.577,A -85,B 0,C 180,E1 -18427.794,E2 -18427.794} C_VEL
LIN {X 0,Y 260.999,Z 337.886,A -85,B 0,C 180,E1 -18429.303,E2 -18429.303} C_VEL
LIN {X 0,Y 259.313,Z 348.076,A -85,B 0,C 180,E1 -18431.021,E2 -18431.021} C_VEL
LIN {X 0,Y 257.617,Z 357.865,A -85,B 0,C 180,E1 -18433.092,E2 -18433.092} C_VEL
LIN {X 0,Y 256.364,Z 366.266,A -85,B 0,C 180,E1 -18435.311,E2 -18435.311} C_VEL
LIN {X 0,Y 255.213,Z 373.422,A -85,B 0,C 180,E1 -18437.677,E2 -18437.677} C_VEL
LIN {X 0,Y 254.508,Z 379.95,A -85,B 0,C 180,E1 -18440.463,E2 -18440.463} C_VEL
LIN {X 0,Y 254.231,Z 384.216,A -85,B 0,C 180,E1 -18442.854,E2 -18442.854} C_VEL
LIN {X 0,Y 254.157,Z 387.367,A -85,B 0,C 180,E1 -18445.241,E2 -18445.241} C_VEL
LIN {X 0,Y 254.216,Z 388.916,A -85,B 0,C 180,E1 -18446.83,E2 -18446.83} C_VEL
LIN {X 0,Y 254.222,Z 389.994,A -85,B 0,C 180,E1 -18448.416,E2 -18448.416} C_VEL
LIN {X 0,Y 254.283,Z 390.644,A -85,B 0,C 180,E1 -18450,E2 -18450} C_VEL
LIN {X 0,Y 254.185,Z 390.881,A -85,B 0,C 180,E1 -18451.584,E2 -18451.584} C_VEL
LIN {X 0,Y 254.128,Z 390.721,A -85,B 0,C 180,E1 -18453.171,E2 -18453.171} C_VEL
LIN {X 0,Y 254.035,Z 389.902,A -85,B 0,C 180,E1 -18455.149,E2 -18455.149} C_VEL
LIN {X 0,Y 254.226,Z 387.703,A -85,B 0,C 180,E1 -18457.945,E2 -18457.945} C_VEL
LIN {X 0,Y 254.702,Z 384.782,A -85,B 0,C 180,E1 -18460.332,E2 -18460.332} C_VEL
LIN {X 0,Y 255.511,Z 380.85,A -85,B 0,C 180,E1 -18462.712,E2 -18462.712} C_VEL
LIN {X 0,Y 256.914,Z 375.816,A -85,B 0,C 180,E1 -18465.063,E2 -18465.063} C_VEL
LIN {X 0,Y 258.636,Z 369.525,A -85,B 0,C 180,E1 -18467.392,E2 -18467.392} C_VEL
LIN {X 0,Y 260.707,Z 361.757,A -85,B 0,C 180,E1 -18469.692,E2 -18469.692} C_VEL
LIN {X 0,Y 262.81,Z 353.857,A -85,B 0,C 180,E1 -18471.574,E2 -18471.574} C_VEL
LIN {X 0,Y 265.4,Z 344.259,A -85,B 0,C 180,E1 -18473.404,E2 -18473.404} C_VEL
LIN {X 0,Y 267.87,Z 333.692,A -85,B 0,C 180,E1 -18475.028,E2 -18475.028} C_VEL
LIN {X 0,Y 270.401,Z 322.006,A -85,B 0,C 180,E1 -18476.429,E2 -18476.429} C_VEL
LIN {X 0,Y 272.559,Z 309.697,A -85,B 0,C 180,E1 -18477.55,E2 -18477.55} C_VEL
LIN {X 0,Y 274.5,Z 296.231,A -85,B 0,C 180,E1 -18478.428,E2 -18478.428} C_VEL
LIN {X 0,Y 275.638,Z 282.782,A -85,B 0,C 180,E1 -18479.015,E2 -18479.015} C_VEL
LIN {X 0,Y 277.905,Z 232.354,A -85,B 0,C 180,E1 -18480.48,E2 -18480.48} C_VEL
LIN {X 0,Y 275.477,Z 212.431,A -85,B 0,C 180,E1 -18481.581,E2 -18481.581} C_VEL
LIN {X 0,Y 273.146,Z 199.196,A -85,B 0,C 180,E1 -18482.46,E2 -18482.46} C_VEL
LIN {X 0,Y 268.123,Z 188.146,A -85,B 0,C 180,E1 -18483.779,E2 -18483.779} C_VEL
LIN {X 0,Y 264.855,Z 181.701,A -85,B 0,C 180,E1 -18484.654,E2 -18484.654} C_VEL
LIN {X 0,Y 261.201,Z 174.424,A -85,B 0,C 180,E1 -18485.719,E2 -18485.719} C_VEL
LIN {X 0,Y 259.2,Z 166.834,A -85,B 0,C 180,E1 -18488.997,E2 -18488.997} C_VEL
LIN {X 0,Y 257.005,Z 159.75,A -85,B 0,C 180,E1 -18492.41,E2 -18492.41} C_VEL
LIN {X 0,Y 256.082,Z 156.591,A -85,B 0,C 180,E1 -18494.066,E2 -18494.066} C_VEL
LIN {X 0,Y 256.088,Z 156.585,A -85,B 0,C 180,E1 -18497.814,E2 -18497.814} C_VEL
LIN {X 0,Y 256.106,Z 156.579,A -85,B 0,C 180,E1 -18500.864,E2 -18500.864} C_VEL
LIN {X 0,Y 256.122,Z 156.578,A -85,B 0,C 180,E1 -18504.813,E2 -18504.813} C_VEL
LIN {X 0,Y 256.092,Z 156.586,A -85,B 0,C 180,E1 -18508.572,E2 -18508.572} C_VEL
LIN {X 0,Y 256.138,Z 156.578,A -85,B 0,C 180,E1 -18512.195,E2 -18512.195} C_VEL
LIN {X 0,Y 256.142,Z 156.577,A -85,B 0,C 180,E1 -18515.696,E2 -18515.696} C_VEL
LIN {X 0,Y 256.162,Z 156.573,A -85,B 0,C 180,E1 -18519.104,E2 -18519.104} C_VEL
LIN {X 0,Y 256.299,Z 156.551,A -85,B 0,C 180,E1 -18524.085,E2 -18524.085} C_VEL
LIN {X 0,Y 256.309,Z 156.548,A -85,B 0,C 180,E1 -18528.934,E2 -18528.934} C_VEL
LIN {X 0,Y 256.539,Z 156.521,A -85,B 0,C 180,E1 -18532.127,E2 -18532.127} C_VEL
LIN {X 0,Y 256.713,Z 156.508,A -85,B 0,C 180,E1 -18538.431,E2 -18538.431} C_VEL
LIN {X 0,Y 256.713,Z 156.508,A -85,B 0,C 180,E1 -18541.568,E2 -18541.568} C_VEL
LIN {X 0,Y 256.47,Z 156.532,A -85,B 0,C 180,E1 -18546.725,E2 -18546.725} C_VEL
LIN {X 0,Y 256.425,Z 156.541,A -85,B 0,C 180,E1 -18549.465,E2 -18549.465} C_VEL
LIN {X 0,Y 256.253,Z 156.563,A -85,B 0,C 180,E1 -18554.29,E2 -18554.29} C_VEL
LIN {X 0,Y 256.285,Z 156.559,A -85,B 0,C 180,E1 -18556.305,E2 -18556.305} C_VEL
LIN {X 0,Y 257.308,Z 159.515,A -85,B 0,C 180,E1 -18556.702,E2 -18556.702} C_VEL
LIN {X 0,Y 259.319,Z 161.953,A -85,B 0,C 180,E1 -18557.253,E2 -18557.253} C_VEL
LIN {X 0,Y 261.468,Z 165.276,A -85,B 0,C 180,E1 -18557.853,E2 -18557.853} C_VEL
LIN {X 0,Y 267.241,Z 174.295,A -85,B 0,C 180,E1 -18559.384,E2 -18559.384} C_VEL
LIN {X 0,Y 272.97,Z 184.235,A -85,B 0,C 180,E1 -18560.814,E2 -18560.814} C_VEL
LIN {X 0,Y 278.395,Z 195.753,A -85,B 0,C 180,E1 -18562.156,E2 -18562.156} C_VEL
LIN {X 0,Y 279.504,Z 198.415,A -85,B 0,C 180,E1 -18562.427,E2 -18562.427} C_VEL
LIN {X 0,Y 276.326,Z 262.499,A -85,B 0,C 180,E1 -18564.287,E2 -18564.287} C_VEL
LIN {X 0,Y 275.085,Z 276.449,A -85,B 0,C 180,E1 -18565.008,E2 -18565.008} C_VEL
LIN {X 0,Y 273.609,Z 288.864,A -85,B 0,C 180,E1 -18565.971,E2 -18565.971} C_VEL
LIN {X 0,Y 271.643,Z 301.19,A -85,B 0,C 180,E1 -18567.255,E2 -18567.255} C_VEL
LIN {X 0,Y 269.623,Z 311.25,A -85,B 0,C 180,E1 -18568.583,E2 -18568.583} C_VEL
LIN {X 0,Y 267.422,Z 321.212,A -85,B 0,C 180,E1 -18570.235,E2 -18570.235} C_VEL
LIN {X 0,Y 264.965,Z 330.561,A -85,B 0,C 180,E1 -18572.161,E2 -18572.161} C_VEL
LIN {X 0,Y 262.729,Z 338.421,A -85,B 0,C 180,E1 -18574.176,E2 -18574.176} C_VEL
LIN {X 0,Y 260.572,Z 345.384,A -85,B 0,C 180,E1 -18576.396,E2 -18576.396} C_VEL
LIN {X 0,Y 258.815,Z 350.967,A -85,B 0,C 180,E1 -18578.649,E2 -18578.649} C_VEL
LIN {X 0,Y 257.352,Z 355.426,A -85,B 0,C 180,E1 -18580.951,E2 -18580.951} C_VEL
LIN {X 0,Y 256.182,Z 358.86,A -85,B 0,C 180,E1 -18583.301,E2 -18583.301} C_VEL
LIN {X 0,Y 255.004,Z 361.896,A -85,B 0,C 180,E1 -18586.449,E2 -18586.449} C_VEL
LIN {X 0,Y 254.529,Z 363.007,A -85,B 0,C 180,E1 -18588.496,E2 -18588.496} C_VEL
LIN {X 0,Y 254.195,Z 363.414,A -85,B 0,C 180,E1 -18590.727,E2 -18590.727} C_VEL
LIN {X 0,Y 254.031,Z 362.906,A -85,B 0,C 180,E1 -18593.351,E2 -18593.351} C_VEL
LIN {X 0,Y 254.218,Z 360.886,A -85,B 0,C 180,E1 -18596.433,E2 -18596.433} C_VEL
LIN {X 0,Y 254.607,Z 358.208,A -85,B 0,C 180,E1 -18598.837,E2 -18598.837} C_VEL
LIN {X 0,Y 255.33,Z 353.55,A -85,B 0,C 180,E1 -18601.739,E2 -18601.739} C_VEL
LIN {X 0,Y 256.193,Z 347.739,A -85,B 0,C 180,E1 -18604.418,E2 -18604.418} C_VEL
LIN {X 0,Y 257.347,Z 341.434,A -85,B 0,C 180,E1 -18606.673,E2 -18606.673} C_VEL
LIN {X 0,Y 258.646,Z 333.709,A -85,B 0,C 180,E1 -18608.898,E2 -18608.898} C_VEL
LIN {X 0,Y 260.277,Z 324.211,A -85,B 0,C 180,E1 -18611.094,E2 -18611.094} C_VEL
LIN {X 0,Y 261.845,Z 313.847,A -85,B 0,C 180,E1 -18613.002,E2 -18613.002} C_VEL
LIN {X 0,Y 263.542,Z 301.906,A -85,B 0,C 180,E1 -18614.732,E2 -18614.732} C_VEL
LIN {X 0,Y 265.014,Z 289.685,A -85,B 0,C 180,E1 -18616.094,E2 -18616.094} C_VEL
LIN {X 0,Y 266.093,Z 277.169,A -85,B 0,C 180,E1 -18617.148,E2 -18617.148} C_VEL
LIN {X 0,Y 267.012,Z 263.921,A -85,B 0,C 180,E1 -18617.929,E2 -18617.929} C_VEL
LIN {X 0,Y 267.65,Z 248.547,A -85,B 0,C 180,E1 -18618.462,E2 -18618.462} C_VEL
LIN {X 0,Y 269.681,Z 189.27,A -85,B 0,C 180,E1 -18620.148,E2 -18620.148} C_VEL
LIN {X 0,Y 264.708,Z 175.968,A -85,B 0,C 180,E1 -18621.024,E2 -18621.024} C_VEL
LIN {X 0,Y 256.627,Z 157.159,A -85,B 0,C 180,E1 -18622.427,E2 -18622.427} C_VEL
LIN {X 0,Y 256.512,Z 156.535,A -85,B 0,C 180,E1 -18622.522,E2 -18622.522} C_VEL
LIN {X 0,Y 256.713,Z 156.507,A -85,B 0,C 180,E1 -18628.431,E2 -18628.431} C_VEL
LIN {X 0,Y 256.713,Z 156.51,A -85,B 0,C 180,E1 -18631.569,E2 -18631.569} C_VEL
LIN {X 0,Y 256.461,Z 156.539,A -85,B 0,C 180,E1 -18636.293,E2 -18636.293} C_VEL
LIN {X 0,Y 256.426,Z 156.544,A -85,B 0,C 180,E1 -18639.465,E2 -18639.465} C_VEL
LIN {X 0,Y 256.232,Z 156.567,A -85,B 0,C 180,E1 -18644.291,E2 -18644.291} C_VEL
LIN {X 0,Y 256.173,Z 156.573,A -85,B 0,C 180,E1 -18647.565,E2 -18647.565} C_VEL
LIN {X 0,Y 256.142,Z 156.578,A -85,B 0,C 180,E1 -18651.111,E2 -18651.111} C_VEL
LIN {X 0,Y 256.171,Z 156.574,A -85,B 0,C 180,E1 -18655.13,E2 -18655.13} C_VEL
LIN {X 0,Y 256.114,Z 156.58,A -85,B 0,C 180,E1 -18659.6,E2 -18659.6} C_VEL
LIN {X 0,Y 256.076,Z 156.585,A -85,B 0,C 180,E1 -18663.291,E2 -18663.291} C_VEL
LIN {X 0,Y 256.113,Z 156.58,A -85,B 0,C 180,E1 -18667.271,E2 -18667.271} C_VEL
LIN {X 0,Y 256.053,Z 156.582,A -85,B 0,C 180,E1 -18671.204,E2 -18671.204} C_VEL
LIN {X 0,Y 256.056,Z 156.588,A -85,B 0,C 180,E1 -18675.53,E2 -18675.53} C_VEL
LIN {X 0,Y 256.053,Z 156.583,A -85,B 0,C 180,E1 -18678.797,E2 -18678.797} C_VEL
LIN {X 0,Y 256.138,Z 156.575,A -85,B 0,C 180,E1 -18682.869,E2 -18682.869} C_VEL
LIN {X 0,Y 256.075,Z 156.584,A -85,B 0,C 180,E1 -18686.709,E2 -18686.709} C_VEL
LIN {X 0,Y 256.103,Z 156.572,A -85,B 0,C 180,E1 -18690.399,E2 -18690.399} C_VEL
LIN {X 0,Y 256.17,Z 156.572,A -85,B 0,C 180,E1 -18694.87,E2 -18694.87} C_VEL
LIN {X 0,Y 256.161,Z 156.574,A -85,B 0,C 180,E1 -18699.105,E2 -18699.105} C_VEL
LIN {X 0,Y 256.299,Z 156.554,A -85,B 0,C 180,E1 -18704.085,E2 -18704.085} C_VEL
LIN {X 0,Y 256.309,Z 156.557,A -85,B 0,C 180,E1 -18708.934,E2 -18708.934} C_VEL
LIN {X 0,Y 256.539,Z 156.52,A -85,B 0,C 180,E1 -18712.127,E2 -18712.127} C_VEL
LIN {X 0,Y 256.714,Z 156.504,A -85,B 0,C 180,E1 -18718.432,E2 -18718.432} C_VEL
LIN {X 0,Y 256.714,Z 156.501,A -85,B 0,C 180,E1 -18721.569,E2 -18721.569} C_VEL
LIN {X 0,Y 256.373,Z 156.541,A -85,B 0,C 180,E1 -18725.35,E2 -18725.35} C_VEL
LIN {X 0,Y 256.111,Z 156.578,A -85,B 0,C 180,E1 -18726.228,E2 -18726.228} C_VEL
LIN {X 0,Y 254.787,Z 156.749,A -85,B 0,C 180,E1 -18727.524,E2 -18727.524} C_VEL
LIN {X 0,Y 250.378,Z 157.295,A -85,B 0,C 180,E1 -18730.54,E2 -18730.54} C_VEL
LIN {X 0,Y 249.298,Z 157.424,A -85,B 0,C 180,E1 -18731.892,E2 -18731.892} C_VEL
LIN {X 0,Y 249.21,Z 157.434,A -85,B 0,C 180,E1 -18732.351,E2 -18732.351} C_VEL
LIN {X 0,Y 249.218,Z 157.442,A -85,B 0,C 180,E1 -18736.504,E2 -18736.504} C_VEL
LIN {X 0,Y 249.084,Z 157.454,A -85,B 0,C 180,E1 -18741.519,E2 -18741.519} C_VEL
LIN {X 0,Y 249.118,Z 157.45,A -85,B 0,C 180,E1 -18745.476,E2 -18745.476} C_VEL
LIN {X 0,Y 249.084,Z 157.458,A -85,B 0,C 180,E1 -18748.994,E2 -18748.994} C_VEL
LIN {X 0,Y 249.037,Z 157.464,A -85,B 0,C 180,E1 -18752.425,E2 -18752.425} C_VEL
LIN {X 0,Y 249.075,Z 157.461,A -85,B 0,C 180,E1 -18756.338,E2 -18756.338} C_VEL
LIN {X 0,Y 249.038,Z 157.464,A -85,B 0,C 180,E1 -18760.472,E2 -18760.472} C_VEL
LIN {X 0,Y 249.009,Z 157.465,A -85,B 0,C 180,E1 -18764.878,E2 -18764.878} C_VEL
LIN {X 0,Y 249.031,Z 157.464,A -85,B 0,C 180,E1 -18767.366,E2 -18767.366} C_VEL
LIN {X 0,Y 249.05,Z 157.465,A -85,B 0,C 180,E1 -18771.624,E2 -18771.624} C_VEL
LIN {X 0,Y 249.128,Z 157.608,A -85,B 0,C 180,E1 -18772.852,E2 -18772.852} C_VEL
LIN {X 0,Y 251.629,Z 168.814,A -85,B 0,C 180,E1 -18776.92,E2 -18776.92} C_VEL
LIN {X 0,Y 253.535,Z 177.936,A -85,B 0,C 180,E1 -18780.069,E2 -18780.069} C_VEL
LIN {X 0,Y 256.295,Z 186.534,A -85,B 0,C 180,E1 -18780.659,E2 -18780.659} C_VEL
LIN {X 0,Y 261.04,Z 223.638,A -85,B 0,C 180,E1 -18782.33,E2 -18782.33} C_VEL
LIN {X 0,Y 261.926,Z 231.634,A -85,B 0,C 180,E1 -18782.667,E2 -18782.667} C_VEL
LIN {X 0,Y 259.962,Z 288.016,A -85,B 0,C 180,E1 -18784.37,E2 -18784.37} C_VEL
LIN {X 0,Y 258.862,Z 302.04,A -85,B 0,C 180,E1 -18785.114,E2 -18785.114} C_VEL
LIN {X 0,Y 257.492,Z 314.034,A -85,B 0,C 180,E1 -18786.046,E2 -18786.046} C_VEL
LIN {X 0,Y 255.83,Z 326.575,A -85,B 0,C 180,E1 -18787.381,E2 -18787.381} C_VEL
LIN {X 0,Y 254.113,Z 337.816,A -85,B 0,C 180,E1 -18788.928,E2 -18788.928} C_VEL
LIN {X 0,Y 252.386,Z 347.934,A -85,B 0,C 180,E1 -18790.691,E2 -18790.691} C_VEL
LIN {X 0,Y 250.712,Z 356.621,A -85,B 0,C 180,E1 -18792.556,E2 -18792.556} C_VEL
LIN {X 0,Y 249.899,Z 362.577,A -85,B 0,C 180,E1 -18794.086,E2 -18794.086} C_VEL
LIN {X 0,Y 248.625,Z 370.384,A -85,B 0,C 180,E1 -18796.514,E2 -18796.514} C_VEL
LIN {X 0,Y 247.832,Z 375.707,A -85,B 0,C 180,E1 -18798.55,E2 -18798.55} C_VEL
LIN {X 0,Y 247.332,Z 380.846,A -85,B 0,C 180,E1 -18801.009,E2 -18801.009} C_VEL
LIN {X 0,Y 247.109,Z 384.797,A -85,B 0,C 180,E1 -18803.468,E2 -18803.468} C_VEL
LIN {X 0,Y 247.071,Z 386.81,A -85,B 0,C 180,E1 -18805.105,E2 -18805.105} C_VEL
LIN {X 0,Y 247.145,Z 388.393,A -85,B 0,C 180,E1 -18806.74,E2 -18806.74} C_VEL
LIN {X 0,Y 247.146,Z 389.529,A -85,B 0,C 180,E1 -18808.37,E2 -18808.37} C_VEL
LIN {X 0,Y 247.201,Z 390.208,A -85,B 0,C 180,E1 -18810,E2 -18810} C_VEL
LIN {X 0,Y 247.109,Z 390.474,A -85,B 0,C 180,E1 -18811.63,E2 -18811.63} C_VEL
LIN {X 0,Y 247.036,Z 390.34,A -85,B 0,C 180,E1 -18813.262,E2 -18813.262} C_VEL
LIN {X 0,Y 246.952,Z 389.696,A -85,B 0,C 180,E1 -18815.081,E2 -18815.081} C_VEL
LIN {X 0,Y 247.165,Z 387.443,A -85,B 0,C 180,E1 -18818.173,E2 -18818.173} C_VEL
LIN {X 0,Y 247.696,Z 384.595,A -85,B 0,C 180,E1 -18820.628,E2 -18820.628} C_VEL
LIN {X 0,Y 248.555,Z 380.735,A -85,B 0,C 180,E1 -18823.073,E2 -18823.073} C_VEL
LIN {X 0,Y 250.047,Z 375.774,A -85,B 0,C 180,E1 -18825.486,E2 -18825.486} C_VEL
LIN {X 0,Y 251.874,Z 369.562,A -85,B 0,C 180,E1 -18827.874,E2 -18827.874} C_VEL
LIN {X 0,Y 254.027,Z 361.892,A -85,B 0,C 180,E1 -18830.232,E2 -18830.232} C_VEL
LIN {X 0,Y 256.224,Z 354.128,A -85,B 0,C 180,E1 -18832.157,E2 -18832.157} C_VEL
LIN {X 0,Y 258.93,Z 344.741,A -85,B 0,C 180,E1 -18834.025,E2 -18834.025} C_VEL
LIN {X 0,Y 261.49,Z 334.398,A -85,B 0,C 180,E1 -18835.682,E2 -18835.682} C_VEL
LIN {X 0,Y 264.101,Z 323.002,A -85,B 0,C 180,E1 -18837.111,E2 -18837.111} C_VEL
LIN {X 0,Y 266.363,Z 311.222,A -85,B 0,C 180,E1 -18838.247,E2 -18838.247} C_VEL
LIN {X 0,Y 268.344,Z 298.402,A -85,B 0,C 180,E1 -18839.142,E2 -18839.142} C_VEL
LIN {X 0,Y 269.756,Z 284.427,A -85,B 0,C 180,E1 -18839.817,E2 -18839.817} C_VEL
LIN {X 0,Y 272.19,Z 233.306,A -85,B 0,C 180,E1 -18841.34,E2 -18841.34} C_VEL
LIN {X 0,Y 269.734,Z 212.679,A -85,B 0,C 180,E1 -18842.534,E2 -18842.534} C_VEL
LIN {X 0,Y 267.927,Z 202.286,A -85,B 0,C 180,E1 -18843.261,E2 -18843.261} C_VEL
LIN {X 0,Y 262.632,Z 190.644,A -85,B 0,C 180,E1 -18844.72,E2 -18844.72} C_VEL
LIN {X 0,Y 258.748,Z 183.069,A -85,B 0,C 180,E1 -18845.834,E2 -18845.834} C_VEL
LIN {X 0,Y 255.895,Z 177.738,A -85,B 0,C 180,E1 -18846.683,E2 -18846.683} C_VEL
LIN {X 0,Y 253.874,Z 173.761,A -85,B 0,C 180,E1 -18847.361,E2 -18847.361} C_VEL
LIN {X 0,Y 251.658,Z 165.892,A -85,B 0,C 180,E1 -18851.059,E2 -18851.059} C_VEL
LIN {X 0,Y 249.87,Z 160.027,A -85,B 0,C 180,E1 -18854.116,E2 -18854.116} C_VEL
LIN {X 0,Y 249.014,Z 157.466,A -85,B 0,C 180,E1 -18855.683,E2 -18855.683} C_VEL
LIN {X 0,Y 249.048,Z 157.466,A -85,B 0,C 180,E1 -18859.634,E2 -18859.634} C_VEL
LIN {X 0,Y 249.076,Z 157.454,A -85,B 0,C 180,E1 -18863.662,E2 -18863.662} C_VEL
LIN {X 0,Y 249.04,Z 157.458,A -85,B 0,C 180,E1 -18867.844,E2 -18867.844} C_VEL
LIN {X 0,Y 249.086,Z 157.452,A -85,B 0,C 180,E1 -18871.337,E2 -18871.337} C_VEL
LIN {X 0,Y 249.134,Z 157.446,A -85,B 0,C 180,E1 -18874.966,E2 -18874.966} C_VEL
LIN {X 0,Y 249.108,Z 157.447,A -85,B 0,C 180,E1 -18880.211,E2 -18880.211} C_VEL
LIN {X 0,Y 249.242,Z 157.434,A -85,B 0,C 180,E1 -18883.621,E2 -18883.621} C_VEL
LIN {X 0,Y 249.252,Z 157.427,A -85,B 0,C 180,E1 -18888.616,E2 -18888.616} C_VEL
LIN {X 0,Y 249.483,Z 157.401,A -85,B 0,C 180,E1 -18891.903,E2 -18891.903} C_VEL
LIN {X 0,Y 249.435,Z 157.406,A -85,B 0,C 180,E1 -18896.769,E2 -18896.769} C_VEL
LIN {X 0,Y 249.727,Z 157.37,A -85,B 0,C 180,E1 -18900,E2 -18900} C_VEL
LIN {X 0,Y 249.434,Z 157.408,A -85,B 0,C 180,E1 -18903.23,E2 -18903.23} C_VEL
LIN {X 0,Y 249.44,Z 157.407,A -85,B 0,C 180,E1 -18906.71,E2 -18906.71} C_VEL
LIN {X 0,Y 249.342,Z 157.425,A -85,B 0,C 180,E1 -18909.736,E2 -18909.736} C_VEL
LIN {X 0,Y 249.221,Z 157.44,A -85,B 0,C 180,E1 -18914.65,E2 -18914.65} C_VEL
LIN {X 0,Y 250.216,Z 160.292,A -85,B 0,C 180,E1 -18915.059,E2 -18915.059} C_VEL
LIN {X 0,Y 252.505,Z 162.932,A -85,B 0,C 180,E1 -18915.746,E2 -18915.746} C_VEL
LIN {X 0,Y 254.666,Z 166.317,A -85,B 0,C 180,E1 -18916.411,E2 -18916.411} C_VEL
LIN {X 0,Y 259.026,Z 172.898,A -85,B 0,C 180,E1 -18917.664,E2 -18917.664} C_VEL
LIN {X 0,Y 265.326,Z 183.147,A -85,B 0,C 180,E1 -18919.375,E2 -18919.375} C_VEL
LIN {X 0,Y 270.189,Z 192.268,A -85,B 0,C 180,E1 -18920.633,E2 -18920.633} C_VEL
LIN {X 0,Y 273.72,Z 200.326,A -85,B 0,C 180,E1 -18921.558,E2 -18921.558} C_VEL
LIN {X 0,Y 270.582,Z 262.63,A -85,B 0,C 180,E1 -18923.419,E2 -18923.419} C_VEL
LIN {X 0,Y 269.364,Z 275.881,A -85,B 0,C 180,E1 -18924.101,E2 -18924.101} C_VEL
LIN {X 0,Y 267.901,Z 287.915,A -85,B 0,C 180,E1 -18925.015,E2 -18925.015} C_VEL
LIN {X 0,Y 266.15,Z 298.94,A -85,B 0,C 180,E1 -18926.129,E2 -18926.129} C_VEL
LIN {X 0,Y 263.752,Z 310.712,A -85,B 0,C 180,E1 -18927.658,E2 -18927.658} C_VEL
LIN {X 0,Y 261.228,Z 321.621,A -85,B 0,C 180,E1 -18929.48,E2 -18929.48} C_VEL
LIN {X 0,Y 258.799,Z 330.423,A -85,B 0,C 180,E1 -18931.32,E2 -18931.32} C_VEL
LIN {X 0,Y 256.571,Z 337.82,A -85,B 0,C 180,E1 -18933.219,E2 -18933.219} C_VEL
